Fanuc TP program (LS listing): FM142654.ls

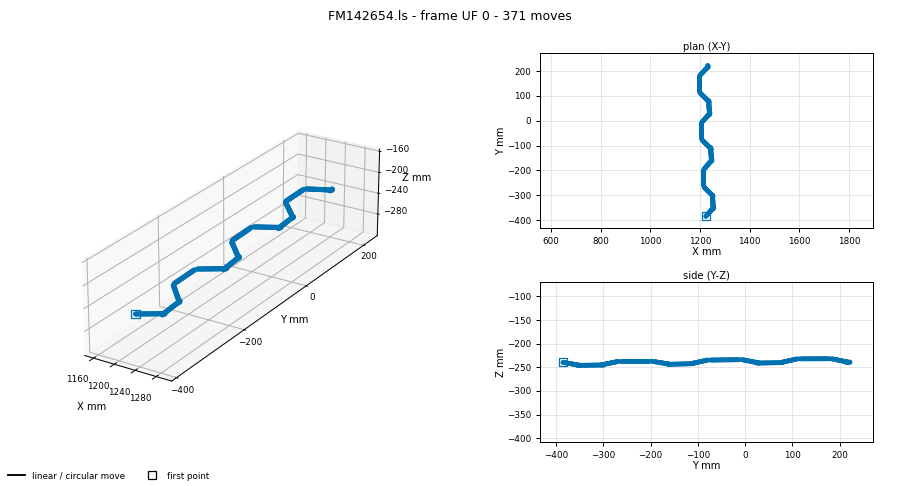
[picture p0: tool path of FM142654.ls in frame UF 0, 371 of 371 moves have a stored position in this frame; points joined in program order, loops and branches not executed]
/PROG  FM142654
/ATTR
OWNER		= MNEDITOR;
COMMENT		= "Auto FANUC move";
PROG_SIZE	= 0;
CREATE		= DATE 26-05-06  TIME 14:26:54;
MODIFIED	= DATE 26-05-06  TIME 14:26:54;
FILE_NAME	= ;
VERSION		= 0;
LINE_COUNT	= 376;
MEMORY_SIZE	= 0;
PROTECT		= READ_WRITE;
TCD:  STACK_SIZE	= 0,
      TASK_PRIORITY	= 50,
      TIME_SLICE	= 0,
      BUSY_LAMP_OFF	= 0,
      ABORT_REQUEST	= 0,
      PAUSE_REQUEST	= 0;
DEFAULT_GROUP	= 1,*,*,*,*;
CONTROL_CODE	= 00000000 00000000;
/MN
   1:  UFRAME_NUM=0 ;
   2:  UTOOL_NUM=1 ;
   3:  R[93]=10 ;
   4:  L P[1] 7mm/sec FINE ;
   5:  L P[2] 7mm/sec CNT50 ;
   6:  L P[3] 7mm/sec CNT50 ;
   7:  L P[4] 7mm/sec CNT50 ;
   8:  L P[5] 7mm/sec CNT50 ;
   9:  L P[6] 7mm/sec CNT50 ;
  10:  L P[7] 7mm/sec CNT50 ;
  11:  L P[8] 7mm/sec CNT50 ;
  12:  L P[9] 7mm/sec CNT50 ;
  13:  L P[10] 7mm/sec CNT50 ;
  14:  L P[11] 7mm/sec CNT50 ;
  15:  L P[12] 7mm/sec CNT50 ;
  16:  L P[13] 7mm/sec CNT50 ;
  17:  L P[14] 7mm/sec CNT50 ;
  18:  L P[15] 7mm/sec CNT50 ;
  19:  L P[16] 7mm/sec CNT50 ;
  20:  L P[17] 7mm/sec CNT50 ;
  21:  L P[18] 7mm/sec CNT50 ;
  22:  L P[19] 7mm/sec CNT50 ;
  23:  L P[20] 7mm/sec CNT50 ;
  24:  L P[21] 7mm/sec CNT50 ;
  25:  L P[22] 7mm/sec CNT50 ;
  26:  L P[23] 7mm/sec CNT50 ;
  27:  L P[24] 7mm/sec CNT50 ;
  28:  L P[25] 7mm/sec CNT50 ;
  29:  L P[26] 7mm/sec CNT50 ;
  30:  L P[27] 7mm/sec CNT50 ;
  31:  L P[28] 7mm/sec CNT50 ;
  32:  L P[29] 7mm/sec CNT50 ;
  33:  L P[30] 7mm/sec CNT50 ;
  34:  L P[31] 7mm/sec CNT50 ;
  35:  L P[32] 7mm/sec CNT50 ;
  36:  L P[33] 7mm/sec CNT50 ;
  37:  L P[34] 7mm/sec CNT50 ;
  38:  L P[35] 7mm/sec CNT50 ;
  39:  L P[36] 7mm/sec CNT50 ;
  40:  L P[37] 7mm/sec CNT50 ;
  41:  L P[38] 7mm/sec CNT50 ;
  42:  L P[39] 7mm/sec CNT50 ;
  43:  L P[40] 7mm/sec CNT50 ;
  44:  L P[41] 7mm/sec CNT50 ;
  45:  L P[42] 7mm/sec CNT50 ;
  46:  L P[43] 7mm/sec CNT50 ;
  47:  L P[44] 7mm/sec CNT50 ;
  48:  L P[45] 7mm/sec CNT50 ;
  49:  L P[46] 7mm/sec CNT50 ;
  50:  L P[47] 7mm/sec CNT50 ;
  51:  L P[48] 7mm/sec CNT50 ;
  52:  L P[49] 7mm/sec CNT50 ;
  53:  L P[50] 7mm/sec CNT50 ;
  54:  L P[51] 7mm/sec CNT50 ;
  55:  L P[52] 7mm/sec CNT50 ;
  56:  L P[53] 7mm/sec CNT50 ;
  57:  L P[54] 7mm/sec CNT50 ;
  58:  L P[55] 7mm/sec CNT50 ;
  59:  L P[56] 7mm/sec CNT50 ;
  60:  L P[57] 7mm/sec CNT50 ;
  61:  L P[58] 7mm/sec CNT50 ;
  62:  L P[59] 7mm/sec CNT50 ;
  63:  L P[60] 7mm/sec CNT50 ;
  64:  L P[61] 7mm/sec CNT50 ;
  65:  L P[62] 7mm/sec CNT50 ;
  66:  L P[63] 7mm/sec CNT50 ;
  67:  L P[64] 7mm/sec CNT50 ;
  68:  L P[65] 7mm/sec CNT50 ;
  69:  L P[66] 7mm/sec CNT50 ;
  70:  L P[67] 7mm/sec CNT50 ;
  71:  L P[68] 7mm/sec CNT50 ;
  72:  L P[69] 7mm/sec CNT50 ;
  73:  L P[70] 7mm/sec CNT50 ;
  74:  L P[71] 7mm/sec CNT50 ;
  75:  L P[72] 7mm/sec CNT50 ;
  76:  L P[73] 7mm/sec CNT50 ;
  77:  L P[74] 7mm/sec CNT50 ;
  78:  L P[75] 7mm/sec CNT50 ;
  79:  L P[76] 7mm/sec CNT50 ;
  80:  L P[77] 7mm/sec CNT50 ;
  81:  L P[78] 7mm/sec CNT50 ;
  82:  L P[79] 7mm/sec CNT50 ;
  83:  L P[80] 7mm/sec CNT50 ;
  84:  L P[81] 7mm/sec CNT50 ;
  85:  L P[82] 7mm/sec CNT50 ;
  86:  L P[83] 7mm/sec CNT50 ;
  87:  L P[84] 7mm/sec CNT50 ;
  88:  L P[85] 7mm/sec CNT50 ;
  89:  L P[86] 7mm/sec CNT50 ;
  90:  L P[87] 7mm/sec CNT50 ;
  91:  L P[88] 7mm/sec CNT50 ;
  92:  L P[89] 7mm/sec CNT50 ;
  93:  L P[90] 7mm/sec CNT50 ;
  94:  L P[91] 7mm/sec CNT50 ;
  95:  L P[92] 7mm/sec CNT50 ;
  96:  L P[93] 7mm/sec CNT50 ;
  97:  L P[94] 7mm/sec CNT50 ;
  98:  L P[95] 7mm/sec CNT50 ;
  99:  L P[96] 7mm/sec CNT50 ;
 100:  L P[97] 7mm/sec CNT50 ;
 101:  L P[98] 7mm/sec CNT50 ;
 102:  L P[99] 7mm/sec CNT50 ;
 103:  L P[100] 7mm/sec CNT50 ;
 104:  L P[101] 7mm/sec CNT50 ;
 105:  L P[102] 7mm/sec CNT50 ;
 106:  L P[103] 7mm/sec CNT50 ;
 107:  L P[104] 7mm/sec CNT50 ;
 108:  L P[105] 7mm/sec CNT50 ;
 109:  L P[106] 7mm/sec CNT50 ;
 110:  L P[107] 7mm/sec CNT50 ;
 111:  L P[108] 7mm/sec CNT50 ;
 112:  L P[109] 7mm/sec CNT50 ;
 113:  L P[110] 7mm/sec CNT50 ;
 114:  L P[111] 7mm/sec CNT50 ;
 115:  L P[112] 7mm/sec CNT50 ;
 116:  L P[113] 7mm/sec CNT50 ;
 117:  L P[114] 7mm/sec CNT50 ;
 118:  L P[115] 7mm/sec CNT50 ;
 119:  L P[116] 7mm/sec CNT50 ;
 120:  L P[117] 7mm/sec CNT50 ;
 121:  L P[118] 7mm/sec CNT50 ;
 122:  L P[119] 7mm/sec CNT50 ;
 123:  L P[120] 7mm/sec CNT50 ;
 124:  L P[121] 7mm/sec CNT50 ;
 125:  L P[122] 7mm/sec CNT50 ;
 126:  L P[123] 7mm/sec CNT50 ;
 127:  L P[124] 7mm/sec CNT50 ;
 128:  L P[125] 7mm/sec CNT50 ;
 129:  L P[126] 7mm/sec CNT50 ;
 130:  L P[127] 7mm/sec CNT50 ;
 131:  L P[128] 7mm/sec CNT50 ;
 132:  L P[129] 7mm/sec CNT50 ;
 133:  L P[130] 7mm/sec CNT50 ;
 134:  L P[131] 7mm/sec CNT50 ;
 135:  L P[132] 7mm/sec CNT50 ;
 136:  L P[133] 7mm/sec CNT50 ;
 137:  L P[134] 7mm/sec CNT50 ;
 138:  L P[135] 7mm/sec CNT50 ;
 139:  L P[136] 7mm/sec CNT50 ;
 140:  L P[137] 7mm/sec CNT50 ;
 141:  L P[138] 7mm/sec CNT50 ;
 142:  L P[139] 7mm/sec CNT50 ;
 143:  L P[140] 7mm/sec CNT50 ;
 144:  L P[141] 7mm/sec CNT50 ;
 145:  L P[142] 7mm/sec CNT50 ;
 146:  L P[143] 7mm/sec CNT50 ;
 147:  L P[144] 7mm/sec CNT50 ;
 148:  L P[145] 7mm/sec CNT50 ;
 149:  L P[146] 7mm/sec CNT50 ;
 150:  L P[147] 7mm/sec CNT50 ;
 151:  L P[148] 7mm/sec CNT50 ;
 152:  L P[149] 7mm/sec CNT50 ;
 153:  L P[150] 7mm/sec CNT50 ;
 154:  L P[151] 7mm/sec CNT50 ;
 155:  L P[152] 7mm/sec CNT50 ;
 156:  L P[153] 7mm/sec CNT50 ;
 157:  L P[154] 7mm/sec CNT50 ;
 158:  L P[155] 7mm/sec CNT50 ;
 159:  L P[156] 7mm/sec CNT50 ;
 160:  L P[157] 7mm/sec CNT50 ;
 161:  L P[158] 7mm/sec CNT50 ;
 162:  L P[159] 7mm/sec CNT50 ;
 163:  L P[160] 7mm/sec CNT50 ;
 164:  L P[161] 7mm/sec CNT50 ;
 165:  L P[162] 7mm/sec CNT50 ;
 166:  L P[163] 7mm/sec CNT50 ;
 167:  L P[164] 7mm/sec CNT50 ;
 168:  L P[165] 7mm/sec CNT50 ;
 169:  L P[166] 7mm/sec CNT50 ;
 170:  L P[167] 7mm/sec CNT50 ;
 171:  L P[168] 7mm/sec CNT50 ;
 172:  L P[169] 7mm/sec CNT50 ;
 173:  L P[170] 7mm/sec CNT50 ;
 174:  L P[171] 7mm/sec CNT50 ;
 175:  L P[172] 7mm/sec CNT50 ;
 176:  L P[173] 7mm/sec CNT50 ;
 177:  L P[174] 7mm/sec CNT50 ;
 178:  L P[175] 7mm/sec CNT50 ;
 179:  L P[176] 7mm/sec CNT50 ;
 180:  L P[177] 7mm/sec CNT50 ;
 181:  L P[178] 7mm/sec CNT50 ;
 182:  L P[179] 7mm/sec CNT50 ;
 183:  L P[180] 7mm/sec CNT50 ;
 184:  L P[181] 7mm/sec CNT50 ;
 185:  L P[182] 7mm/sec CNT50 ;
 186:  L P[183] 7mm/sec CNT50 ;
 187:  L P[184] 7mm/sec CNT50 ;
 188:  L P[185] 7mm/sec CNT50 ;
 189:  L P[186] 7mm/sec CNT50 ;
 190:  L P[187] 7mm/sec CNT50 ;
 191:  L P[188] 7mm/sec CNT50 ;
 192:  L P[189] 7mm/sec CNT50 ;
 193:  L P[190] 7mm/sec CNT50 ;
 194:  L P[191] 7mm/sec CNT50 ;
 195:  L P[192] 7mm/sec CNT50 ;
 196:  L P[193] 7mm/sec CNT50 ;
 197:  L P[194] 7mm/sec CNT50 ;
 198:  L P[195] 7mm/sec CNT50 ;
 199:  L P[196] 7mm/sec CNT50 ;
 200:  L P[197] 7mm/sec CNT50 ;
 201:  L P[198] 7mm/sec CNT50 ;
 202:  L P[199] 7mm/sec CNT50 ;
 203:  L P[200] 7mm/sec CNT50 ;
 204:  L P[201] 7mm/sec CNT50 ;
 205:  L P[202] 7mm/sec CNT50 ;
 206:  L P[203] 7mm/sec CNT50 ;
 207:  L P[204] 7mm/sec CNT50 ;
 208:  L P[205] 7mm/sec CNT50 ;
 209:  L P[206] 7mm/sec CNT50 ;
 210:  L P[207] 7mm/sec CNT50 ;
 211:  L P[208] 7mm/sec CNT50 ;
 212:  L P[209] 7mm/sec CNT50 ;
 213:  L P[210] 7mm/sec CNT50 ;
 214:  L P[211] 7mm/sec CNT50 ;
 215:  L P[212] 7mm/sec CNT50 ;
 216:  L P[213] 7mm/sec CNT50 ;
 217:  L P[214] 7mm/sec CNT50 ;
 218:  L P[215] 7mm/sec CNT50 ;
 219:  L P[216] 7mm/sec CNT50 ;
 220:  L P[217] 7mm/sec CNT50 ;
 221:  L P[218] 7mm/sec CNT50 ;
 222:  L P[219] 7mm/sec CNT50 ;
 223:  L P[220] 7mm/sec CNT50 ;
 224:  L P[221] 7mm/sec CNT50 ;
 225:  L P[222] 7mm/sec CNT50 ;
 226:  L P[223] 7mm/sec CNT50 ;
 227:  L P[224] 7mm/sec CNT50 ;
 228:  L P[225] 7mm/sec CNT50 ;
 229:  L P[226] 7mm/sec CNT50 ;
 230:  L P[227] 7mm/sec CNT50 ;
 231:  L P[228] 7mm/sec CNT50 ;
 232:  L P[229] 7mm/sec CNT50 ;
 233:  L P[230] 7mm/sec CNT50 ;
 234:  L P[231] 7mm/sec CNT50 ;
 235:  L P[232] 7mm/sec CNT50 ;
 236:  L P[233] 7mm/sec CNT50 ;
 237:  L P[234] 7mm/sec CNT50 ;
 238:  L P[235] 7mm/sec CNT50 ;
 239:  L P[236] 7mm/sec CNT50 ;
 240:  L P[237] 7mm/sec CNT50 ;
 241:  L P[238] 7mm/sec CNT50 ;
 242:  L P[239] 7mm/sec CNT50 ;
 243:  L P[240] 7mm/sec CNT50 ;
 244:  L P[241] 7mm/sec CNT50 ;
 245:  L P[242] 7mm/sec CNT50 ;
 246:  L P[243] 7mm/sec CNT50 ;
 247:  L P[244] 7mm/sec CNT50 ;
 248:  L P[245] 7mm/sec CNT50 ;
 249:  L P[246] 7mm/sec CNT50 ;
 250:  L P[247] 7mm/sec CNT50 ;
 251:  L P[248] 7mm/sec CNT50 ;
 252:  L P[249] 7mm/sec CNT50 ;
 253:  L P[250] 7mm/sec CNT50 ;
 254:  L P[251] 7mm/sec CNT50 ;
 255:  L P[252] 7mm/sec CNT50 ;
 256:  L P[253] 7mm/sec CNT50 ;
 257:  L P[254] 7mm/sec CNT50 ;
 258:  L P[255] 7mm/sec CNT50 ;
 259:  L P[256] 7mm/sec CNT50 ;
 260:  L P[257] 7mm/sec CNT50 ;
 261:  L P[258] 7mm/sec CNT50 ;
 262:  L P[259] 7mm/sec CNT50 ;
 263:  L P[260] 7mm/sec CNT50 ;
 264:  L P[261] 7mm/sec CNT50 ;
 265:  L P[262] 7mm/sec CNT50 ;
 266:  L P[263] 7mm/sec CNT50 ;
 267:  L P[264] 7mm/sec CNT50 ;
 268:  L P[265] 7mm/sec CNT50 ;
 269:  L P[266] 7mm/sec CNT50 ;
 270:  L P[267] 7mm/sec CNT50 ;
 271:  L P[268] 7mm/sec CNT50 ;
 272:  L P[269] 7mm/sec CNT50 ;
 273:  L P[270] 7mm/sec CNT50 ;
 274:  L P[271] 7mm/sec CNT50 ;
 275:  L P[272] 7mm/sec CNT50 ;
 276:  L P[273] 7mm/sec CNT50 ;
 277:  L P[274] 7mm/sec CNT50 ;
 278:  L P[275] 7mm/sec CNT50 ;
 279:  L P[276] 7mm/sec CNT50 ;
 280:  L P[277] 7mm/sec CNT50 ;
 281:  L P[278] 7mm/sec CNT50 ;
 282:  L P[279] 7mm/sec CNT50 ;
 283:  L P[280] 7mm/sec CNT50 ;
 284:  L P[281] 7mm/sec CNT50 ;
 285:  L P[282] 7mm/sec CNT50 ;
 286:  L P[283] 7mm/sec CNT50 ;
 287:  L P[284] 7mm/sec CNT50 ;
 288:  L P[285] 7mm/sec CNT50 ;
 289:  L P[286] 7mm/sec CNT50 ;
 290:  L P[287] 7mm/sec CNT50 ;
 291:  L P[288] 7mm/sec CNT50 ;
 292:  L P[289] 7mm/sec CNT50 ;
 293:  L P[290] 7mm/sec CNT50 ;
 294:  L P[291] 7mm/sec CNT50 ;
 295:  L P[292] 7mm/sec CNT50 ;
 296:  L P[293] 7mm/sec CNT50 ;
 297:  L P[294] 7mm/sec CNT50 ;
 298:  L P[295] 7mm/sec CNT50 ;
 299:  L P[296] 7mm/sec CNT50 ;
 300:  L P[297] 7mm/sec CNT50 ;
 301:  L P[298] 7mm/sec CNT50 ;
 302:  L P[299] 7mm/sec CNT50 ;
 303:  L P[300] 7mm/sec CNT50 ;
 304:  L P[301] 7mm/sec CNT50 ;
 305:  L P[302] 7mm/sec CNT50 ;
 306:  L P[303] 7mm/sec CNT50 ;
 307:  L P[304] 7mm/sec CNT50 ;
 308:  L P[305] 7mm/sec CNT50 ;
 309:  L P[306] 7mm/sec CNT50 ;
 310:  L P[307] 7mm/sec CNT50 ;
 311:  L P[308] 7mm/sec CNT50 ;
 312:  L P[309] 7mm/sec CNT50 ;
 313:  L P[310] 7mm/sec CNT50 ;
 314:  L P[311] 7mm/sec CNT50 ;
 315:  L P[312] 7mm/sec CNT50 ;
 316:  L P[313] 7mm/sec CNT50 ;
 317:  L P[314] 7mm/sec CNT50 ;
 318:  L P[315] 7mm/sec CNT50 ;
 319:  L P[316] 7mm/sec CNT50 ;
 320:  L P[317] 7mm/sec CNT50 ;
 321:  L P[318] 7mm/sec CNT50 ;
 322:  L P[319] 7mm/sec CNT50 ;
 323:  L P[320] 7mm/sec CNT50 ;
 324:  L P[321] 7mm/sec CNT50 ;
 325:  L P[322] 7mm/sec CNT50 ;
 326:  L P[323] 7mm/sec CNT50 ;
 327:  L P[324] 7mm/sec CNT50 ;
 328:  L P[325] 7mm/sec CNT50 ;
 329:  L P[326] 7mm/sec CNT50 ;
 330:  L P[327] 7mm/sec CNT50 ;
 331:  L P[328] 7mm/sec CNT50 ;
 332:  L P[329] 7mm/sec CNT50 ;
 333:  L P[330] 7mm/sec CNT50 ;
 334:  L P[331] 7mm/sec CNT50 ;
 335:  L P[332] 7mm/sec CNT50 ;
 336:  L P[333] 7mm/sec CNT50 ;
 337:  L P[334] 7mm/sec CNT50 ;
 338:  L P[335] 7mm/sec CNT50 ;
 339:  L P[336] 7mm/sec CNT50 ;
 340:  L P[337] 7mm/sec CNT50 ;
 341:  L P[338] 7mm/sec CNT50 ;
 342:  L P[339] 7mm/sec CNT50 ;
 343:  L P[340] 7mm/sec CNT50 ;
 344:  L P[341] 7mm/sec CNT50 ;
 345:  L P[342] 7mm/sec CNT50 ;
 346:  L P[343] 7mm/sec CNT50 ;
 347:  L P[344] 7mm/sec CNT50 ;
 348:  L P[345] 7mm/sec CNT50 ;
 349:  L P[346] 7mm/sec CNT50 ;
 350:  L P[347] 7mm/sec CNT50 ;
 351:  L P[348] 7mm/sec CNT50 ;
 352:  L P[349] 7mm/sec CNT50 ;
 353:  L P[350] 7mm/sec CNT50 ;
 354:  L P[351] 7mm/sec CNT50 ;
 355:  L P[352] 7mm/sec CNT50 ;
 356:  L P[353] 7mm/sec CNT50 ;
 357:  L P[354] 7mm/sec CNT50 ;
 358:  L P[355] 7mm/sec CNT50 ;
 359:  L P[356] 7mm/sec CNT50 ;
 360:  L P[357] 7mm/sec CNT50 ;
 361:  L P[358] 7mm/sec CNT50 ;
 362:  L P[359] 7mm/sec CNT50 ;
 363:  L P[360] 7mm/sec CNT50 ;
 364:  L P[361] 7mm/sec CNT50 ;
 365:  L P[362] 7mm/sec CNT50 ;
 366:  L P[363] 7mm/sec CNT50 ;
 367:  L P[364] 7mm/sec CNT50 ;
 368:  L P[365] 7mm/sec CNT50 ;
 369:  L P[366] 7mm/sec CNT50 ;
 370:  L P[367] 7mm/sec CNT50 ;
 371:  L P[368] 7mm/sec CNT50 ;
 372:  L P[369] 7mm/sec CNT50 ;
 373:  L P[370] 7mm/sec CNT50 ;
 374:  L P[371] 7mm/sec FINE ;
 375:  R[93]=1 ;
 376:  END ;
/POS
P[1]{
   GP1:
	UF : 0, UT : 1,		CONFIG : 'N U T, 0, 0, 0',
	X = 1223.194  mm,	Y = -385.306  mm,	Z = -239.653  mm,
	W = 0.000 deg,	P = 30.000 deg,	R = 138.708 deg
};
P[2]{
   GP1:
	UF : 0, UT : 1,		CONFIG : 'N U T, 0, 0, 0',
	X = 1224.503  mm,	Y = -383.816  mm,	Z = -239.910  mm,
	W = 0.000 deg,	P = 30.000 deg,	R = 138.708 deg
};
P[3]{
   GP1:
	UF : 0, UT : 1,		CONFIG : 'N U T, 0, 0, 0',
	X = 1225.812  mm,	Y = -382.326  mm,	Z = -240.167  mm,
	W = 0.000 deg,	P = 30.000 deg,	R = 138.708 deg
};
P[4]{
   GP1:
	UF : 0, UT : 1,		CONFIG : 'N U T, 0, 0, 0',
	X = 1227.120  mm,	Y = -380.835  mm,	Z = -240.424  mm,
	W = 0.000 deg,	P = 30.000 deg,	R = 138.708 deg
};
P[5]{
   GP1:
	UF : 0, UT : 1,		CONFIG : 'N U T, 0, 0, 0',
	X = 1228.429  mm,	Y = -379.345  mm,	Z = -240.682  mm,
	W = 0.000 deg,	P = 30.000 deg,	R = 138.708 deg
};
P[6]{
   GP1:
	UF : 0, UT : 1,		CONFIG : 'N U T, 0, 0, 0',
	X = 1229.738  mm,	Y = -377.855  mm,	Z = -240.939  mm,
	W = 0.000 deg,	P = 30.000 deg,	R = 138.708 deg
};
P[7]{
   GP1:
	UF : 0, UT : 1,		CONFIG : 'N U T, 0, 0, 0',
	X = 1231.047  mm,	Y = -376.365  mm,	Z = -241.196  mm,
	W = 0.000 deg,	P = 30.000 deg,	R = 138.708 deg
};
P[8]{
   GP1:
	UF : 0, UT : 1,		CONFIG : 'N U T, 0, 0, 0',
	X = 1232.356  mm,	Y = -374.874  mm,	Z = -241.453  mm,
	W = 0.000 deg,	P = 30.000 deg,	R = 138.708 deg
};
P[9]{
   GP1:
	UF : 0, UT : 1,		CONFIG : 'N U T, 0, 0, 0',
	X = 1233.665  mm,	Y = -373.384  mm,	Z = -241.710  mm,
	W = 0.000 deg,	P = 30.000 deg,	R = 138.708 deg
};
P[10]{
   GP1:
	UF : 0, UT : 1,		CONFIG : 'N U T, 0, 0, 0',
	X = 1234.973  mm,	Y = -371.894  mm,	Z = -241.967  mm,
	W = 0.000 deg,	P = 30.000 deg,	R = 138.708 deg
};
P[11]{
   GP1:
	UF : 0, UT : 1,		CONFIG : 'N U T, 0, 0, 0',
	X = 1236.282  mm,	Y = -370.404  mm,	Z = -242.225  mm,
	W = 0.000 deg,	P = 30.000 deg,	R = 138.708 deg
};
P[12]{
   GP1:
	UF : 0, UT : 1,		CONFIG : 'N U T, 0, 0, 0',
	X = 1237.591  mm,	Y = -368.913  mm,	Z = -242.482  mm,
	W = 0.000 deg,	P = 30.000 deg,	R = 138.708 deg
};
P[13]{
   GP1:
	UF : 0, UT : 1,		CONFIG : 'N U T, 0, 0, 0',
	X = 1238.900  mm,	Y = -367.423  mm,	Z = -242.739  mm,
	W = 0.000 deg,	P = 30.000 deg,	R = 138.708 deg
};
P[14]{
   GP1:
	UF : 0, UT : 1,		CONFIG : 'N U T, 0, 0, 0',
	X = 1240.209  mm,	Y = -365.933  mm,	Z = -242.996  mm,
	W = 0.000 deg,	P = 30.000 deg,	R = 138.708 deg
};
P[15]{
   GP1:
	UF : 0, UT : 1,		CONFIG : 'N U T, 0, 0, 0',
	X = 1241.518  mm,	Y = -364.443  mm,	Z = -243.253  mm,
	W = 0.000 deg,	P = 30.000 deg,	R = 138.708 deg
};
P[16]{
   GP1:
	UF : 0, UT : 1,		CONFIG : 'N U T, 0, 0, 0',
	X = 1242.826  mm,	Y = -362.952  mm,	Z = -243.510  mm,
	W = 0.000 deg,	P = 30.000 deg,	R = 138.708 deg
};
P[17]{
   GP1:
	UF : 0, UT : 1,		CONFIG : 'N U T, 0, 0, 0',
	X = 1244.135  mm,	Y = -361.462  mm,	Z = -243.767  mm,
	W = 0.000 deg,	P = 30.000 deg,	R = 138.708 deg
};
P[18]{
   GP1:
	UF : 0, UT : 1,		CONFIG : 'N U T, 0, 0, 0',
	X = 1245.444  mm,	Y = -359.972  mm,	Z = -244.025  mm,
	W = 0.000 deg,	P = 30.000 deg,	R = 138.708 deg
};
P[19]{
   GP1:
	UF : 0, UT : 1,		CONFIG : 'N U T, 0, 0, 0',
	X = 1246.753  mm,	Y = -358.482  mm,	Z = -244.282  mm,
	W = 0.000 deg,	P = 30.000 deg,	R = 138.708 deg
};
P[20]{
   GP1:
	UF : 0, UT : 1,		CONFIG : 'N U T, 0, 0, 0',
	X = 1248.062  mm,	Y = -356.991  mm,	Z = -244.539  mm,
	W = 0.000 deg,	P = 30.000 deg,	R = 138.708 deg
};
P[21]{
   GP1:
	UF : 0, UT : 1,		CONFIG : 'N U T, 0, 0, 0',
	X = 1249.371  mm,	Y = -355.501  mm,	Z = -244.796  mm,
	W = 0.000 deg,	P = 30.000 deg,	R = 147.583 deg
};
P[22]{
   GP1:
	UF : 0, UT : 1,		CONFIG : 'N U T, 0, 0, 0',
	X = 1250.679  mm,	Y = -354.011  mm,	Z = -245.053  mm,
	W = 0.000 deg,	P = 30.000 deg,	R = 156.458 deg
};
P[23]{
   GP1:
	UF : 0, UT : 1,		CONFIG : 'N U T, 0, 0, 0',
	X = 1251.988  mm,	Y = -352.521  mm,	Z = -245.310  mm,
	W = 0.000 deg,	P = 30.000 deg,	R = 165.333 deg
};
P[24]{
   GP1:
	UF : 0, UT : 1,		CONFIG : 'N U T, 0, 0, 0',
	X = 1253.297  mm,	Y = -351.030  mm,	Z = -245.568  mm,
	W = 0.000 deg,	P = 30.000 deg,	R = 174.208 deg
};
P[25]{
   GP1:
	UF : 0, UT : 1,		CONFIG : 'N U T, 0, 0, 0',
	X = 1254.606  mm,	Y = -349.540  mm,	Z = -245.825  mm,
	W = 0.000 deg,	P = 30.000 deg,	R = -176.917 deg
};
P[26]{
   GP1:
	UF : 0, UT : 1,		CONFIG : 'N U T, 0, 0, 0',
	X = 1254.120  mm,	Y = -350.543  mm,	Z = -245.999  mm,
	W = 0.000 deg,	P = 30.000 deg,	R = -176.917 deg
};
P[27]{
   GP1:
	UF : 0, UT : 1,		CONFIG : 'N U T, 0, 0, 0',
	X = 1252.987  mm,	Y = -355.024  mm,	Z = -245.989  mm,
	W = 0.000 deg,	P = 30.000 deg,	R = -176.917 deg
};
P[28]{
   GP1:
	UF : 0, UT : 1,		CONFIG : 'N U T, 0, 0, 0',
	X = 1252.879  mm,	Y = -353.027  mm,	Z = -245.958  mm,
	W = 0.000 deg,	P = 30.000 deg,	R = -176.917 deg
};
P[29]{
   GP1:
	UF : 0, UT : 1,		CONFIG : 'N U T, 0, 0, 0',
	X = 1252.772  mm,	Y = -351.030  mm,	Z = -245.926  mm,
	W = 0.000 deg,	P = 30.000 deg,	R = -176.917 deg
};
P[30]{
   GP1:
	UF : 0, UT : 1,		CONFIG : 'N U T, 0, 0, 0',
	X = 1252.664  mm,	Y = -349.033  mm,	Z = -245.895  mm,
	W = 0.000 deg,	P = 30.000 deg,	R = -176.917 deg
};
P[31]{
   GP1:
	UF : 0, UT : 1,		CONFIG : 'N U T, 0, 0, 0',
	X = 1252.557  mm,	Y = -347.036  mm,	Z = -245.863  mm,
	W = 0.000 deg,	P = 30.000 deg,	R = -176.917 deg
};
P[32]{
   GP1:
	UF : 0, UT : 1,		CONFIG : 'N U T, 0, 0, 0',
	X = 1252.449  mm,	Y = -345.039  mm,	Z = -245.832  mm,
	W = 0.000 deg,	P = 30.000 deg,	R = -176.917 deg
};
P[33]{
   GP1:
	UF : 0, UT : 1,		CONFIG : 'N U T, 0, 0, 0',
	X = 1252.342  mm,	Y = -343.042  mm,	Z = -245.801  mm,
	W = 0.000 deg,	P = 30.000 deg,	R = -176.917 deg
};
P[34]{
   GP1:
	UF : 0, UT : 1,		CONFIG : 'N U T, 0, 0, 0',
	X = 1252.234  mm,	Y = -341.046  mm,	Z = -245.769  mm,
	W = 0.000 deg,	P = 30.000 deg,	R = -176.917 deg
};
P[35]{
   GP1:
	UF : 0, UT : 1,		CONFIG : 'N U T, 0, 0, 0',
	X = 1252.126  mm,	Y = -339.049  mm,	Z = -245.738  mm,
	W = 0.000 deg,	P = 30.000 deg,	R = -176.917 deg
};
P[36]{
   GP1:
	UF : 0, UT : 1,		CONFIG : 'N U T, 0, 0, 0',
	X = 1252.019  mm,	Y = -337.052  mm,	Z = -245.706  mm,
	W = 0.000 deg,	P = 30.000 deg,	R = -176.917 deg
};
P[37]{
   GP1:
	UF : 0, UT : 1,		CONFIG : 'N U T, 0, 0, 0',
	X = 1251.911  mm,	Y = -335.055  mm,	Z = -245.675  mm,
	W = 0.000 deg,	P = 30.000 deg,	R = -176.917 deg
};
P[38]{
   GP1:
	UF : 0, UT : 1,		CONFIG : 'N U T, 0, 0, 0',
	X = 1251.804  mm,	Y = -333.058  mm,	Z = -245.644  mm,
	W = 0.000 deg,	P = 30.000 deg,	R = -176.917 deg
};
P[39]{
   GP1:
	UF : 0, UT : 1,		CONFIG : 'N U T, 0, 0, 0',
	X = 1251.696  mm,	Y = -331.061  mm,	Z = -245.612  mm,
	W = 0.000 deg,	P = 30.000 deg,	R = -176.917 deg
};
P[40]{
   GP1:
	UF : 0, UT : 1,		CONFIG : 'N U T, 0, 0, 0',
	X = 1251.589  mm,	Y = -329.064  mm,	Z = -245.581  mm,
	W = 0.000 deg,	P = 30.000 deg,	R = -176.917 deg
};
P[41]{
   GP1:
	UF : 0, UT : 1,		CONFIG : 'N U T, 0, 0, 0',
	X = 1251.481  mm,	Y = -327.068  mm,	Z = -245.549  mm,
	W = 0.000 deg,	P = 30.000 deg,	R = -176.917 deg
};
P[42]{
   GP1:
	UF : 0, UT : 1,		CONFIG : 'N U T, 0, 0, 0',
	X = 1251.374  mm,	Y = -325.071  mm,	Z = -245.518  mm,
	W = 0.000 deg,	P = 30.000 deg,	R = -176.917 deg
};
P[43]{
   GP1:
	UF : 0, UT : 1,		CONFIG : 'N U T, 0, 0, 0',
	X = 1251.266  mm,	Y = -323.074  mm,	Z = -245.487  mm,
	W = 0.000 deg,	P = 30.000 deg,	R = -176.917 deg
};
P[44]{
   GP1:
	UF : 0, UT : 1,		CONFIG : 'N U T, 0, 0, 0',
	X = 1251.158  mm,	Y = -321.077  mm,	Z = -245.455  mm,
	W = 0.000 deg,	P = 30.000 deg,	R = -176.917 deg
};
P[45]{
   GP1:
	UF : 0, UT : 1,		CONFIG : 'N U T, 0, 0, 0',
	X = 1251.051  mm,	Y = -319.080  mm,	Z = -245.424  mm,
	W = 0.000 deg,	P = 30.000 deg,	R = -176.917 deg
};
P[46]{
   GP1:
	UF : 0, UT : 1,		CONFIG : 'N U T, 0, 0, 0',
	X = 1250.943  mm,	Y = -317.083  mm,	Z = -245.392  mm,
	W = 0.000 deg,	P = 30.000 deg,	R = -176.917 deg
};
P[47]{
   GP1:
	UF : 0, UT : 1,		CONFIG : 'N U T, 0, 0, 0',
	X = 1250.836  mm,	Y = -315.086  mm,	Z = -245.361  mm,
	W = 0.000 deg,	P = 30.000 deg,	R = -176.917 deg
};
P[48]{
   GP1:
	UF : 0, UT : 1,		CONFIG : 'N U T, 0, 0, 0',
	X = 1250.728  mm,	Y = -313.090  mm,	Z = -245.329  mm,
	W = 0.000 deg,	P = 30.000 deg,	R = -176.917 deg
};
P[49]{
   GP1:
	UF : 0, UT : 1,		CONFIG : 'N U T, 0, 0, 0',
	X = 1250.621  mm,	Y = -311.093  mm,	Z = -245.298  mm,
	W = 0.000 deg,	P = 30.000 deg,	R = -176.917 deg
};
P[50]{
   GP1:
	UF : 0, UT : 1,		CONFIG : 'N U T, 0, 0, 0',
	X = 1250.513  mm,	Y = -309.096  mm,	Z = -245.267  mm,
	W = 0.000 deg,	P = 30.000 deg,	R = -176.917 deg
};
P[51]{
   GP1:
	UF : 0, UT : 1,		CONFIG : 'N U T, 0, 0, 0',
	X = 1250.405  mm,	Y = -307.099  mm,	Z = -245.235  mm,
	W = 0.000 deg,	P = 30.000 deg,	R = -165.910 deg
};
P[52]{
   GP1:
	UF : 0, UT : 1,		CONFIG : 'N U T, 0, 0, 0',
	X = 1250.298  mm,	Y = -305.102  mm,	Z = -245.204  mm,
	W = 0.000 deg,	P = 30.000 deg,	R = -157.583 deg
};
P[53]{
   GP1:
	UF : 0, UT : 1,		CONFIG : 'N U T, 0, 0, 0',
	X = 1250.190  mm,	Y = -303.105  mm,	Z = -245.172  mm,
	W = 0.000 deg,	P = 30.000 deg,	R = -149.255 deg
};
P[54]{
   GP1:
	UF : 0, UT : 1,		CONFIG : 'N U T, 0, 0, 0',
	X = 1250.083  mm,	Y = -301.108  mm,	Z = -245.141  mm,
	W = 0.000 deg,	P = 30.000 deg,	R = -140.928 deg
};
P[55]{
   GP1:
	UF : 0, UT : 1,		CONFIG : 'N U T, 0, 0, 0',
	X = 1249.975  mm,	Y = -299.112  mm,	Z = -245.110  mm,
	W = 0.000 deg,	P = 30.000 deg,	R = -135.281 deg
};
P[56]{
   GP1:
	UF : 0, UT : 1,		CONFIG : 'N U T, 0, 0, 0',
	X = 1250.851  mm,	Y = -301.869  mm,	Z = -245.095  mm,
	W = 0.000 deg,	P = 30.000 deg,	R = -135.281 deg
};
P[57]{
   GP1:
	UF : 0, UT : 1,		CONFIG : 'N U T, 0, 0, 0',
	X = 1252.068  mm,	Y = -303.926  mm,	Z = -244.940  mm,
	W = 0.000 deg,	P = 30.000 deg,	R = -135.281 deg
};
P[58]{
   GP1:
	UF : 0, UT : 1,		CONFIG : 'N U T, 0, 0, 0',
	X = 1250.676  mm,	Y = -302.520  mm,	Z = -244.647  mm,
	W = 0.000 deg,	P = 30.000 deg,	R = -135.281 deg
};
P[59]{
   GP1:
	UF : 0, UT : 1,		CONFIG : 'N U T, 0, 0, 0',
	X = 1249.283  mm,	Y = -301.114  mm,	Z = -244.355  mm,
	W = 0.000 deg,	P = 30.000 deg,	R = -135.281 deg
};
P[60]{
   GP1:
	UF : 0, UT : 1,		CONFIG : 'N U T, 0, 0, 0',
	X = 1247.891  mm,	Y = -299.708  mm,	Z = -244.062  mm,
	W = 0.000 deg,	P = 30.000 deg,	R = -135.281 deg
};
P[61]{
   GP1:
	UF : 0, UT : 1,		CONFIG : 'N U T, 0, 0, 0',
	X = 1246.499  mm,	Y = -298.303  mm,	Z = -243.770  mm,
	W = 0.000 deg,	P = 30.000 deg,	R = -135.281 deg
};
P[62]{
   GP1:
	UF : 0, UT : 1,		CONFIG : 'N U T, 0, 0, 0',
	X = 1245.107  mm,	Y = -296.897  mm,	Z = -243.477  mm,
	W = 0.000 deg,	P = 30.000 deg,	R = -135.281 deg
};
P[63]{
   GP1:
	UF : 0, UT : 1,		CONFIG : 'N U T, 0, 0, 0',
	X = 1243.715  mm,	Y = -295.491  mm,	Z = -243.185  mm,
	W = 0.000 deg,	P = 30.000 deg,	R = -135.281 deg
};
P[64]{
   GP1:
	UF : 0, UT : 1,		CONFIG : 'N U T, 0, 0, 0',
	X = 1242.323  mm,	Y = -294.085  mm,	Z = -242.892  mm,
	W = 0.000 deg,	P = 30.000 deg,	R = -135.281 deg
};
P[65]{
   GP1:
	UF : 0, UT : 1,		CONFIG : 'N U T, 0, 0, 0',
	X = 1240.931  mm,	Y = -292.679  mm,	Z = -242.599  mm,
	W = 0.000 deg,	P = 30.000 deg,	R = -135.281 deg
};
P[66]{
   GP1:
	UF : 0, UT : 1,		CONFIG : 'N U T, 0, 0, 0',
	X = 1239.539  mm,	Y = -291.273  mm,	Z = -242.307  mm,
	W = 0.000 deg,	P = 30.000 deg,	R = -135.281 deg
};
P[67]{
   GP1:
	UF : 0, UT : 1,		CONFIG : 'N U T, 0, 0, 0',
	X = 1238.146  mm,	Y = -289.867  mm,	Z = -242.014  mm,
	W = 0.000 deg,	P = 30.000 deg,	R = -135.281 deg
};
P[68]{
   GP1:
	UF : 0, UT : 1,		CONFIG : 'N U T, 0, 0, 0',
	X = 1236.754  mm,	Y = -288.462  mm,	Z = -241.722  mm,
	W = 0.000 deg,	P = 30.000 deg,	R = -135.281 deg
};
P[69]{
   GP1:
	UF : 0, UT : 1,		CONFIG : 'N U T, 0, 0, 0',
	X = 1235.362  mm,	Y = -287.056  mm,	Z = -241.429  mm,
	W = 0.000 deg,	P = 30.000 deg,	R = -135.281 deg
};
P[70]{
   GP1:
	UF : 0, UT : 1,		CONFIG : 'N U T, 0, 0, 0',
	X = 1233.970  mm,	Y = -285.650  mm,	Z = -241.137  mm,
	W = 0.000 deg,	P = 30.000 deg,	R = -135.281 deg
};
P[71]{
   GP1:
	UF : 0, UT : 1,		CONFIG : 'N U T, 0, 0, 0',
	X = 1232.578  mm,	Y = -284.244  mm,	Z = -240.844  mm,
	W = 0.000 deg,	P = 30.000 deg,	R = -135.281 deg
};
P[72]{
   GP1:
	UF : 0, UT : 1,		CONFIG : 'N U T, 0, 0, 0',
	X = 1231.186  mm,	Y = -282.838  mm,	Z = -240.551  mm,
	W = 0.000 deg,	P = 30.000 deg,	R = -135.281 deg
};
P[73]{
   GP1:
	UF : 0, UT : 1,		CONFIG : 'N U T, 0, 0, 0',
	X = 1229.794  mm,	Y = -281.432  mm,	Z = -240.259  mm,
	W = 0.000 deg,	P = 30.000 deg,	R = -135.281 deg
};
P[74]{
   GP1:
	UF : 0, UT : 1,		CONFIG : 'N U T, 0, 0, 0',
	X = 1228.402  mm,	Y = -280.026  mm,	Z = -239.966  mm,
	W = 0.000 deg,	P = 30.000 deg,	R = -135.281 deg
};
P[75]{
   GP1:
	UF : 0, UT : 1,		CONFIG : 'N U T, 0, 0, 0',
	X = 1227.010  mm,	Y = -278.621  mm,	Z = -239.674  mm,
	W = 0.000 deg,	P = 30.000 deg,	R = -135.281 deg
};
P[76]{
   GP1:
	UF : 0, UT : 1,		CONFIG : 'N U T, 0, 0, 0',
	X = 1225.617  mm,	Y = -277.215  mm,	Z = -239.381  mm,
	W = 0.000 deg,	P = 30.000 deg,	R = -135.281 deg
};
P[77]{
   GP1:
	UF : 0, UT : 1,		CONFIG : 'N U T, 0, 0, 0',
	X = 1224.225  mm,	Y = -275.809  mm,	Z = -239.089  mm,
	W = 0.000 deg,	P = 30.000 deg,	R = -139.912 deg
};
P[78]{
   GP1:
	UF : 0, UT : 1,		CONFIG : 'N U T, 0, 0, 0',
	X = 1222.833  mm,	Y = -274.403  mm,	Z = -238.796  mm,
	W = 0.000 deg,	P = 30.000 deg,	R = -148.662 deg
};
P[79]{
   GP1:
	UF : 0, UT : 1,		CONFIG : 'N U T, 0, 0, 0',
	X = 1221.441  mm,	Y = -272.997  mm,	Z = -238.503  mm,
	W = 0.000 deg,	P = 30.000 deg,	R = -157.411 deg
};
P[80]{
   GP1:
	UF : 0, UT : 1,		CONFIG : 'N U T, 0, 0, 0',
	X = 1220.049  mm,	Y = -271.591  mm,	Z = -238.211  mm,
	W = 0.000 deg,	P = 30.000 deg,	R = -166.161 deg
};
P[81]{
   GP1:
	UF : 0, UT : 1,		CONFIG : 'N U T, 0, 0, 0',
	X = 1218.657  mm,	Y = -270.186  mm,	Z = -237.918  mm,
	W = 0.000 deg,	P = 30.000 deg,	R = -174.911 deg
};
P[82]{
   GP1:
	UF : 0, UT : 1,		CONFIG : 'N U T, 0, 0, 0',
	X = 1216.735  mm,	Y = -268.155  mm,	Z = -237.671  mm,
	W = 0.000 deg,	P = 30.000 deg,	R = -179.030 deg
};
P[83]{
   GP1:
	UF : 0, UT : 1,		CONFIG : 'N U T, 0, 0, 0',
	X = 1214.582  mm,	Y = -261.821  mm,	Z = -237.670  mm,
	W = 0.000 deg,	P = 30.000 deg,	R = -179.030 deg
};
P[84]{
   GP1:
	UF : 0, UT : 1,		CONFIG : 'N U T, 0, 0, 0',
	X = 1214.549  mm,	Y = -259.821  mm,	Z = -237.662  mm,
	W = 0.000 deg,	P = 30.000 deg,	R = -179.030 deg
};
P[85]{
   GP1:
	UF : 0, UT : 1,		CONFIG : 'N U T, 0, 0, 0',
	X = 1214.515  mm,	Y = -257.821  mm,	Z = -237.655  mm,
	W = 0.000 deg,	P = 30.000 deg,	R = -179.030 deg
};
P[86]{
   GP1:
	UF : 0, UT : 1,		CONFIG : 'N U T, 0, 0, 0',
	X = 1214.481  mm,	Y = -255.822  mm,	Z = -237.648  mm,
	W = 0.000 deg,	P = 30.000 deg,	R = -179.030 deg
};
P[87]{
   GP1:
	UF : 0, UT : 1,		CONFIG : 'N U T, 0, 0, 0',
	X = 1214.447  mm,	Y = -253.822  mm,	Z = -237.640  mm,
	W = 0.000 deg,	P = 30.000 deg,	R = -179.030 deg
};
P[88]{
   GP1:
	UF : 0, UT : 1,		CONFIG : 'N U T, 0, 0, 0',
	X = 1214.413  mm,	Y = -251.822  mm,	Z = -237.633  mm,
	W = 0.000 deg,	P = 30.000 deg,	R = -179.030 deg
};
P[89]{
   GP1:
	UF : 0, UT : 1,		CONFIG : 'N U T, 0, 0, 0',
	X = 1214.379  mm,	Y = -249.822  mm,	Z = -237.625  mm,
	W = 0.000 deg,	P = 30.000 deg,	R = -179.030 deg
};
P[90]{
   GP1:
	UF : 0, UT : 1,		CONFIG : 'N U T, 0, 0, 0',
	X = 1214.345  mm,	Y = -247.823  mm,	Z = -237.618  mm,
	W = 0.000 deg,	P = 30.000 deg,	R = -179.030 deg
};
P[91]{
   GP1:
	UF : 0, UT : 1,		CONFIG : 'N U T, 0, 0, 0',
	X = 1214.311  mm,	Y = -245.823  mm,	Z = -237.610  mm,
	W = 0.000 deg,	P = 30.000 deg,	R = -179.030 deg
};
P[92]{
   GP1:
	UF : 0, UT : 1,		CONFIG : 'N U T, 0, 0, 0',
	X = 1214.278  mm,	Y = -243.823  mm,	Z = -237.603  mm,
	W = 0.000 deg,	P = 30.000 deg,	R = -179.030 deg
};
P[93]{
   GP1:
	UF : 0, UT : 1,		CONFIG : 'N U T, 0, 0, 0',
	X = 1214.244  mm,	Y = -241.824  mm,	Z = -237.595  mm,
	W = 0.000 deg,	P = 30.000 deg,	R = -179.030 deg
};
P[94]{
   GP1:
	UF : 0, UT : 1,		CONFIG : 'N U T, 0, 0, 0',
	X = 1214.210  mm,	Y = -239.824  mm,	Z = -237.588  mm,
	W = 0.000 deg,	P = 30.000 deg,	R = -179.030 deg
};
P[95]{
   GP1:
	UF : 0, UT : 1,		CONFIG : 'N U T, 0, 0, 0',
	X = 1214.176  mm,	Y = -237.824  mm,	Z = -237.581  mm,
	W = 0.000 deg,	P = 30.000 deg,	R = -179.030 deg
};
P[96]{
   GP1:
	UF : 0, UT : 1,		CONFIG : 'N U T, 0, 0, 0',
	X = 1214.142  mm,	Y = -235.825  mm,	Z = -237.573  mm,
	W = 0.000 deg,	P = 30.000 deg,	R = -179.030 deg
};
P[97]{
   GP1:
	UF : 0, UT : 1,		CONFIG : 'N U T, 0, 0, 0',
	X = 1214.108  mm,	Y = -233.825  mm,	Z = -237.566  mm,
	W = 0.000 deg,	P = 30.000 deg,	R = -179.030 deg
};
P[98]{
   GP1:
	UF : 0, UT : 1,		CONFIG : 'N U T, 0, 0, 0',
	X = 1214.074  mm,	Y = -231.825  mm,	Z = -237.558  mm,
	W = 0.000 deg,	P = 30.000 deg,	R = -179.030 deg
};
P[99]{
   GP1:
	UF : 0, UT : 1,		CONFIG : 'N U T, 0, 0, 0',
	X = 1214.041  mm,	Y = -229.826  mm,	Z = -237.551  mm,
	W = 0.000 deg,	P = 30.000 deg,	R = -179.030 deg
};
P[100]{
   GP1:
	UF : 0, UT : 1,		CONFIG : 'N U T, 0, 0, 0',
	X = 1214.007  mm,	Y = -227.826  mm,	Z = -237.543  mm,
	W = 0.000 deg,	P = 30.000 deg,	R = -179.030 deg
};
P[101]{
   GP1:
	UF : 0, UT : 1,		CONFIG : 'N U T, 0, 0, 0',
	X = 1213.973  mm,	Y = -225.826  mm,	Z = -237.536  mm,
	W = 0.000 deg,	P = 30.000 deg,	R = -179.030 deg
};
P[102]{
   GP1:
	UF : 0, UT : 1,		CONFIG : 'N U T, 0, 0, 0',
	X = 1213.939  mm,	Y = -223.826  mm,	Z = -237.528  mm,
	W = 0.000 deg,	P = 30.000 deg,	R = -179.030 deg
};
P[103]{
   GP1:
	UF : 0, UT : 1,		CONFIG : 'N U T, 0, 0, 0',
	X = 1213.905  mm,	Y = -221.827  mm,	Z = -237.521  mm,
	W = 0.000 deg,	P = 30.000 deg,	R = -179.030 deg
};
P[104]{
   GP1:
	UF : 0, UT : 1,		CONFIG : 'N U T, 0, 0, 0',
	X = 1213.871  mm,	Y = -219.827  mm,	Z = -237.514  mm,
	W = 0.000 deg,	P = 30.000 deg,	R = -179.030 deg
};
P[105]{
   GP1:
	UF : 0, UT : 1,		CONFIG : 'N U T, 0, 0, 0',
	X = 1213.837  mm,	Y = -217.827  mm,	Z = -237.506  mm,
	W = 0.000 deg,	P = 30.000 deg,	R = -179.030 deg
};
P[106]{
   GP1:
	UF : 0, UT : 1,		CONFIG : 'N U T, 0, 0, 0',
	X = 1213.803  mm,	Y = -215.828  mm,	Z = -237.499  mm,
	W = 0.000 deg,	P = 30.000 deg,	R = -179.030 deg
};
P[107]{
   GP1:
	UF : 0, UT : 1,		CONFIG : 'N U T, 0, 0, 0',
	X = 1213.770  mm,	Y = -213.828  mm,	Z = -237.491  mm,
	W = 0.000 deg,	P = 30.000 deg,	R = -179.030 deg
};
P[108]{
   GP1:
	UF : 0, UT : 1,		CONFIG : 'N U T, 0, 0, 0',
	X = 1213.736  mm,	Y = -211.828  mm,	Z = -237.484  mm,
	W = 0.000 deg,	P = 30.000 deg,	R = -179.030 deg
};
P[109]{
   GP1:
	UF : 0, UT : 1,		CONFIG : 'N U T, 0, 0, 0',
	X = 1213.702  mm,	Y = -209.829  mm,	Z = -237.476  mm,
	W = 0.000 deg,	P = 30.000 deg,	R = 171.466 deg
};
P[110]{
   GP1:
	UF : 0, UT : 1,		CONFIG : 'N U T, 0, 0, 0',
	X = 1213.668  mm,	Y = -207.829  mm,	Z = -237.469  mm,
	W = 0.000 deg,	P = 30.000 deg,	R = 163.237 deg
};
P[111]{
   GP1:
	UF : 0, UT : 1,		CONFIG : 'N U T, 0, 0, 0',
	X = 1213.634  mm,	Y = -205.829  mm,	Z = -237.461  mm,
	W = 0.000 deg,	P = 30.000 deg,	R = 155.008 deg
};
P[112]{
   GP1:
	UF : 0, UT : 1,		CONFIG : 'N U T, 0, 0, 0',
	X = 1213.600  mm,	Y = -203.829  mm,	Z = -237.454  mm,
	W = 0.000 deg,	P = 30.000 deg,	R = 146.778 deg
};
P[113]{
   GP1:
	UF : 0, UT : 1,		CONFIG : 'N U T, 0, 0, 0',
	X = 1213.600  mm,	Y = -201.160  mm,	Z = -237.448  mm,
	W = 0.000 deg,	P = 30.000 deg,	R = 139.825 deg
};
P[114]{
   GP1:
	UF : 0, UT : 1,		CONFIG : 'N U T, 0, 0, 0',
	X = 1216.110  mm,	Y = -195.277  mm,	Z = -237.483  mm,
	W = 0.000 deg,	P = 30.000 deg,	R = 139.825 deg
};
P[115]{
   GP1:
	UF : 0, UT : 1,		CONFIG : 'N U T, 0, 0, 0',
	X = 1217.390  mm,	Y = -193.761  mm,	Z = -237.733  mm,
	W = 0.000 deg,	P = 30.000 deg,	R = 139.825 deg
};
P[116]{
   GP1:
	UF : 0, UT : 1,		CONFIG : 'N U T, 0, 0, 0',
	X = 1218.670  mm,	Y = -192.245  mm,	Z = -237.983  mm,
	W = 0.000 deg,	P = 30.000 deg,	R = 139.825 deg
};
P[117]{
   GP1:
	UF : 0, UT : 1,		CONFIG : 'N U T, 0, 0, 0',
	X = 1219.950  mm,	Y = -190.729  mm,	Z = -238.232  mm,
	W = 0.000 deg,	P = 30.000 deg,	R = 139.825 deg
};
P[118]{
   GP1:
	UF : 0, UT : 1,		CONFIG : 'N U T, 0, 0, 0',
	X = 1221.230  mm,	Y = -189.213  mm,	Z = -238.482  mm,
	W = 0.000 deg,	P = 30.000 deg,	R = 139.825 deg
};
P[119]{
   GP1:
	UF : 0, UT : 1,		CONFIG : 'N U T, 0, 0, 0',
	X = 1222.510  mm,	Y = -187.696  mm,	Z = -238.732  mm,
	W = 0.000 deg,	P = 30.000 deg,	R = 139.825 deg
};
P[120]{
   GP1:
	UF : 0, UT : 1,		CONFIG : 'N U T, 0, 0, 0',
	X = 1223.790  mm,	Y = -186.180  mm,	Z = -238.982  mm,
	W = 0.000 deg,	P = 30.000 deg,	R = 139.825 deg
};
P[121]{
   GP1:
	UF : 0, UT : 1,		CONFIG : 'N U T, 0, 0, 0',
	X = 1225.071  mm,	Y = -184.664  mm,	Z = -239.232  mm,
	W = 0.000 deg,	P = 30.000 deg,	R = 139.825 deg
};
P[122]{
   GP1:
	UF : 0, UT : 1,		CONFIG : 'N U T, 0, 0, 0',
	X = 1226.351  mm,	Y = -183.148  mm,	Z = -239.482  mm,
	W = 0.000 deg,	P = 30.000 deg,	R = 139.825 deg
};
P[123]{
   GP1:
	UF : 0, UT : 1,		CONFIG : 'N U T, 0, 0, 0',
	X = 1227.631  mm,	Y = -181.632  mm,	Z = -239.732  mm,
	W = 0.000 deg,	P = 30.000 deg,	R = 139.825 deg
};
P[124]{
   GP1:
	UF : 0, UT : 1,		CONFIG : 'N U T, 0, 0, 0',
	X = 1228.911  mm,	Y = -180.116  mm,	Z = -239.982  mm,
	W = 0.000 deg,	P = 30.000 deg,	R = 139.825 deg
};
P[125]{
   GP1:
	UF : 0, UT : 1,		CONFIG : 'N U T, 0, 0, 0',
	X = 1230.191  mm,	Y = -178.599  mm,	Z = -240.232  mm,
	W = 0.000 deg,	P = 30.000 deg,	R = 139.825 deg
};
P[126]{
   GP1:
	UF : 0, UT : 1,		CONFIG : 'N U T, 0, 0, 0',
	X = 1231.471  mm,	Y = -177.083  mm,	Z = -240.481  mm,
	W = 0.000 deg,	P = 30.000 deg,	R = 139.825 deg
};
P[127]{
   GP1:
	UF : 0, UT : 1,		CONFIG : 'N U T, 0, 0, 0',
	X = 1232.751  mm,	Y = -175.567  mm,	Z = -240.731  mm,
	W = 0.000 deg,	P = 30.000 deg,	R = 139.825 deg
};
P[128]{
   GP1:
	UF : 0, UT : 1,		CONFIG : 'N U T, 0, 0, 0',
	X = 1234.032  mm,	Y = -174.051  mm,	Z = -240.981  mm,
	W = 0.000 deg,	P = 30.000 deg,	R = 139.825 deg
};
P[129]{
   GP1:
	UF : 0, UT : 1,		CONFIG : 'N U T, 0, 0, 0',
	X = 1235.312  mm,	Y = -172.535  mm,	Z = -241.231  mm,
	W = 0.000 deg,	P = 30.000 deg,	R = 139.825 deg
};
P[130]{
   GP1:
	UF : 0, UT : 1,		CONFIG : 'N U T, 0, 0, 0',
	X = 1236.592  mm,	Y = -171.019  mm,	Z = -241.481  mm,
	W = 0.000 deg,	P = 30.000 deg,	R = 139.825 deg
};
P[131]{
   GP1:
	UF : 0, UT : 1,		CONFIG : 'N U T, 0, 0, 0',
	X = 1237.872  mm,	Y = -169.502  mm,	Z = -241.731  mm,
	W = 0.000 deg,	P = 30.000 deg,	R = 139.825 deg
};
P[132]{
   GP1:
	UF : 0, UT : 1,		CONFIG : 'N U T, 0, 0, 0',
	X = 1239.152  mm,	Y = -167.986  mm,	Z = -241.981  mm,
	W = 0.000 deg,	P = 30.000 deg,	R = 139.825 deg
};
P[133]{
   GP1:
	UF : 0, UT : 1,		CONFIG : 'N U T, 0, 0, 0',
	X = 1240.432  mm,	Y = -166.470  mm,	Z = -242.231  mm,
	W = 0.000 deg,	P = 30.000 deg,	R = 139.825 deg
};
P[134]{
   GP1:
	UF : 0, UT : 1,		CONFIG : 'N U T, 0, 0, 0',
	X = 1241.712  mm,	Y = -164.954  mm,	Z = -242.480  mm,
	W = 0.000 deg,	P = 30.000 deg,	R = 141.055 deg
};
P[135]{
   GP1:
	UF : 0, UT : 1,		CONFIG : 'N U T, 0, 0, 0',
	X = 1242.993  mm,	Y = -163.438  mm,	Z = -242.730  mm,
	W = 0.000 deg,	P = 30.000 deg,	R = 149.779 deg
};
P[136]{
   GP1:
	UF : 0, UT : 1,		CONFIG : 'N U T, 0, 0, 0',
	X = 1244.273  mm,	Y = -161.921  mm,	Z = -242.980  mm,
	W = 0.000 deg,	P = 30.000 deg,	R = 158.503 deg
};
P[137]{
   GP1:
	UF : 0, UT : 1,		CONFIG : 'N U T, 0, 0, 0',
	X = 1245.553  mm,	Y = -160.405  mm,	Z = -243.230  mm,
	W = 0.000 deg,	P = 30.000 deg,	R = 167.226 deg
};
P[138]{
   GP1:
	UF : 0, UT : 1,		CONFIG : 'N U T, 0, 0, 0',
	X = 1246.833  mm,	Y = -158.889  mm,	Z = -243.480  mm,
	W = 0.000 deg,	P = 30.000 deg,	R = 175.950 deg
};
P[139]{
   GP1:
	UF : 0, UT : 1,		CONFIG : 'N U T, 0, 0, 0',
	X = 1248.113  mm,	Y = -157.373  mm,	Z = -243.730  mm,
	W = 0.000 deg,	P = 30.000 deg,	R = -176.557 deg
};
P[140]{
   GP1:
	UF : 0, UT : 1,		CONFIG : 'N U T, 0, 0, 0',
	X = 1245.929  mm,	Y = -163.288  mm,	Z = -243.763  mm,
	W = 0.000 deg,	P = 30.000 deg,	R = -176.557 deg
};
P[141]{
   GP1:
	UF : 0, UT : 1,		CONFIG : 'N U T, 0, 0, 0',
	X = 1245.837  mm,	Y = -162.492  mm,	Z = -243.720  mm,
	W = 0.000 deg,	P = 30.000 deg,	R = -176.557 deg
};
P[142]{
   GP1:
	UF : 0, UT : 1,		CONFIG : 'N U T, 0, 0, 0',
	X = 1245.717  mm,	Y = -160.496  mm,	Z = -243.670  mm,
	W = 0.000 deg,	P = 30.000 deg,	R = -176.557 deg
};
P[143]{
   GP1:
	UF : 0, UT : 1,		CONFIG : 'N U T, 0, 0, 0',
	X = 1245.597  mm,	Y = -158.501  mm,	Z = -243.621  mm,
	W = 0.000 deg,	P = 30.000 deg,	R = -176.557 deg
};
P[144]{
   GP1:
	UF : 0, UT : 1,		CONFIG : 'N U T, 0, 0, 0',
	X = 1245.477  mm,	Y = -156.505  mm,	Z = -243.571  mm,
	W = 0.000 deg,	P = 30.000 deg,	R = -176.557 deg
};
P[145]{
   GP1:
	UF : 0, UT : 1,		CONFIG : 'N U T, 0, 0, 0',
	X = 1245.357  mm,	Y = -154.509  mm,	Z = -243.522  mm,
	W = 0.000 deg,	P = 30.000 deg,	R = -176.557 deg
};
P[146]{
   GP1:
	UF : 0, UT : 1,		CONFIG : 'N U T, 0, 0, 0',
	X = 1245.237  mm,	Y = -152.513  mm,	Z = -243.472  mm,
	W = 0.000 deg,	P = 30.000 deg,	R = -176.557 deg
};
P[147]{
   GP1:
	UF : 0, UT : 1,		CONFIG : 'N U T, 0, 0, 0',
	X = 1245.117  mm,	Y = -150.518  mm,	Z = -243.422  mm,
	W = 0.000 deg,	P = 30.000 deg,	R = -176.557 deg
};
P[148]{
   GP1:
	UF : 0, UT : 1,		CONFIG : 'N U T, 0, 0, 0',
	X = 1244.997  mm,	Y = -148.522  mm,	Z = -243.373  mm,
	W = 0.000 deg,	P = 30.000 deg,	R = -176.557 deg
};
P[149]{
   GP1:
	UF : 0, UT : 1,		CONFIG : 'N U T, 0, 0, 0',
	X = 1244.876  mm,	Y = -146.526  mm,	Z = -243.323  mm,
	W = 0.000 deg,	P = 30.000 deg,	R = -176.557 deg
};
P[150]{
   GP1:
	UF : 0, UT : 1,		CONFIG : 'N U T, 0, 0, 0',
	X = 1244.756  mm,	Y = -144.530  mm,	Z = -243.274  mm,
	W = 0.000 deg,	P = 30.000 deg,	R = -176.557 deg
};
P[151]{
   GP1:
	UF : 0, UT : 1,		CONFIG : 'N U T, 0, 0, 0',
	X = 1244.636  mm,	Y = -142.534  mm,	Z = -243.224  mm,
	W = 0.000 deg,	P = 30.000 deg,	R = -176.557 deg
};
P[152]{
   GP1:
	UF : 0, UT : 1,		CONFIG : 'N U T, 0, 0, 0',
	X = 1244.516  mm,	Y = -140.539  mm,	Z = -243.175  mm,
	W = 0.000 deg,	P = 30.000 deg,	R = -176.557 deg
};
P[153]{
   GP1:
	UF : 0, UT : 1,		CONFIG : 'N U T, 0, 0, 0',
	X = 1244.396  mm,	Y = -138.543  mm,	Z = -243.125  mm,
	W = 0.000 deg,	P = 30.000 deg,	R = -176.557 deg
};
P[154]{
   GP1:
	UF : 0, UT : 1,		CONFIG : 'N U T, 0, 0, 0',
	X = 1244.276  mm,	Y = -136.547  mm,	Z = -243.076  mm,
	W = 0.000 deg,	P = 30.000 deg,	R = -176.557 deg
};
P[155]{
   GP1:
	UF : 0, UT : 1,		CONFIG : 'N U T, 0, 0, 0',
	X = 1244.156  mm,	Y = -134.551  mm,	Z = -243.026  mm,
	W = 0.000 deg,	P = 30.000 deg,	R = -176.557 deg
};
P[156]{
   GP1:
	UF : 0, UT : 1,		CONFIG : 'N U T, 0, 0, 0',
	X = 1244.036  mm,	Y = -132.556  mm,	Z = -242.976  mm,
	W = 0.000 deg,	P = 30.000 deg,	R = -176.557 deg
};
P[157]{
   GP1:
	UF : 0, UT : 1,		CONFIG : 'N U T, 0, 0, 0',
	X = 1243.916  mm,	Y = -130.560  mm,	Z = -242.927  mm,
	W = 0.000 deg,	P = 30.000 deg,	R = -176.557 deg
};
P[158]{
   GP1:
	UF : 0, UT : 1,		CONFIG : 'N U T, 0, 0, 0',
	X = 1243.796  mm,	Y = -128.564  mm,	Z = -242.877  mm,
	W = 0.000 deg,	P = 30.000 deg,	R = -176.557 deg
};
P[159]{
   GP1:
	UF : 0, UT : 1,		CONFIG : 'N U T, 0, 0, 0',
	X = 1243.676  mm,	Y = -126.568  mm,	Z = -242.828  mm,
	W = 0.000 deg,	P = 30.000 deg,	R = -176.557 deg
};
P[160]{
   GP1:
	UF : 0, UT : 1,		CONFIG : 'N U T, 0, 0, 0',
	X = 1243.556  mm,	Y = -124.572  mm,	Z = -242.778  mm,
	W = 0.000 deg,	P = 30.000 deg,	R = -176.557 deg
};
P[161]{
   GP1:
	UF : 0, UT : 1,		CONFIG : 'N U T, 0, 0, 0',
	X = 1243.436  mm,	Y = -122.577  mm,	Z = -242.729  mm,
	W = 0.000 deg,	P = 30.000 deg,	R = -176.557 deg
};
P[162]{
   GP1:
	UF : 0, UT : 1,		CONFIG : 'N U T, 0, 0, 0',
	X = 1243.316  mm,	Y = -120.581  mm,	Z = -242.679  mm,
	W = 0.000 deg,	P = 30.000 deg,	R = -176.557 deg
};
P[163]{
   GP1:
	UF : 0, UT : 1,		CONFIG : 'N U T, 0, 0, 0',
	X = 1243.196  mm,	Y = -118.585  mm,	Z = -242.630  mm,
	W = 0.000 deg,	P = 30.000 deg,	R = -176.557 deg
};
P[164]{
   GP1:
	UF : 0, UT : 1,		CONFIG : 'N U T, 0, 0, 0',
	X = 1243.076  mm,	Y = -116.589  mm,	Z = -242.580  mm,
	W = 0.000 deg,	P = 30.000 deg,	R = -169.254 deg
};
P[165]{
   GP1:
	UF : 0, UT : 1,		CONFIG : 'N U T, 0, 0, 0',
	X = 1242.956  mm,	Y = -114.594  mm,	Z = -242.530  mm,
	W = 0.000 deg,	P = 30.000 deg,	R = -160.840 deg
};
P[166]{
   GP1:
	UF : 0, UT : 1,		CONFIG : 'N U T, 0, 0, 0',
	X = 1242.835  mm,	Y = -112.598  mm,	Z = -242.481  mm,
	W = 0.000 deg,	P = 30.000 deg,	R = -152.425 deg
};
P[167]{
   GP1:
	UF : 0, UT : 1,		CONFIG : 'N U T, 0, 0, 0',
	X = 1242.715  mm,	Y = -110.602  mm,	Z = -242.431  mm,
	W = 0.000 deg,	P = 30.000 deg,	R = -144.010 deg
};
P[168]{
   GP1:
	UF : 0, UT : 1,		CONFIG : 'N U T, 0, 0, 0',
	X = 1242.595  mm,	Y = -108.606  mm,	Z = -242.382  mm,
	W = 0.000 deg,	P = 30.000 deg,	R = -135.595 deg
};
P[169]{
   GP1:
	UF : 0, UT : 1,		CONFIG : 'N U T, 0, 0, 0',
	X = 1244.490  mm,	Y = -113.472  mm,	Z = -242.371  mm,
	W = 0.000 deg,	P = 30.000 deg,	R = -134.483 deg
};
P[170]{
   GP1:
	UF : 0, UT : 1,		CONFIG : 'N U T, 0, 0, 0',
	X = 1244.451  mm,	Y = -113.616  mm,	Z = -242.141  mm,
	W = 0.000 deg,	P = 30.000 deg,	R = -134.483 deg
};
P[171]{
   GP1:
	UF : 0, UT : 1,		CONFIG : 'N U T, 0, 0, 0',
	X = 1243.040  mm,	Y = -112.230  mm,	Z = -241.845  mm,
	W = 0.000 deg,	P = 30.000 deg,	R = -134.483 deg
};
P[172]{
   GP1:
	UF : 0, UT : 1,		CONFIG : 'N U T, 0, 0, 0',
	X = 1241.629  mm,	Y = -110.845  mm,	Z = -241.548  mm,
	W = 0.000 deg,	P = 30.000 deg,	R = -134.483 deg
};
P[173]{
   GP1:
	UF : 0, UT : 1,		CONFIG : 'N U T, 0, 0, 0',
	X = 1240.218  mm,	Y = -109.459  mm,	Z = -241.252  mm,
	W = 0.000 deg,	P = 30.000 deg,	R = -134.483 deg
};
P[174]{
   GP1:
	UF : 0, UT : 1,		CONFIG : 'N U T, 0, 0, 0',
	X = 1238.807  mm,	Y = -108.073  mm,	Z = -240.955  mm,
	W = 0.000 deg,	P = 30.000 deg,	R = -134.483 deg
};
P[175]{
   GP1:
	UF : 0, UT : 1,		CONFIG : 'N U T, 0, 0, 0',
	X = 1237.396  mm,	Y = -106.687  mm,	Z = -240.659  mm,
	W = 0.000 deg,	P = 30.000 deg,	R = -134.483 deg
};
P[176]{
   GP1:
	UF : 0, UT : 1,		CONFIG : 'N U T, 0, 0, 0',
	X = 1235.985  mm,	Y = -105.301  mm,	Z = -240.362  mm,
	W = 0.000 deg,	P = 30.000 deg,	R = -134.483 deg
};
P[177]{
   GP1:
	UF : 0, UT : 1,		CONFIG : 'N U T, 0, 0, 0',
	X = 1234.573  mm,	Y = -103.915  mm,	Z = -240.066  mm,
	W = 0.000 deg,	P = 30.000 deg,	R = -134.483 deg
};
P[178]{
   GP1:
	UF : 0, UT : 1,		CONFIG : 'N U T, 0, 0, 0',
	X = 1233.162  mm,	Y = -102.529  mm,	Z = -239.769  mm,
	W = 0.000 deg,	P = 30.000 deg,	R = -134.483 deg
};
P[179]{
   GP1:
	UF : 0, UT : 1,		CONFIG : 'N U T, 0, 0, 0',
	X = 1231.751  mm,	Y = -101.143  mm,	Z = -239.473  mm,
	W = 0.000 deg,	P = 30.000 deg,	R = -134.483 deg
};
P[180]{
   GP1:
	UF : 0, UT : 1,		CONFIG : 'N U T, 0, 0, 0',
	X = 1230.340  mm,	Y = -99.757  mm,	Z = -239.176  mm,
	W = 0.000 deg,	P = 30.000 deg,	R = -134.483 deg
};
P[181]{
   GP1:
	UF : 0, UT : 1,		CONFIG : 'N U T, 0, 0, 0',
	X = 1228.929  mm,	Y = -98.371  mm,	Z = -238.880  mm,
	W = 0.000 deg,	P = 30.000 deg,	R = -134.483 deg
};
P[182]{
   GP1:
	UF : 0, UT : 1,		CONFIG : 'N U T, 0, 0, 0',
	X = 1227.518  mm,	Y = -96.985  mm,	Z = -238.583  mm,
	W = 0.000 deg,	P = 30.000 deg,	R = -134.483 deg
};
P[183]{
   GP1:
	UF : 0, UT : 1,		CONFIG : 'N U T, 0, 0, 0',
	X = 1226.107  mm,	Y = -95.600  mm,	Z = -238.287  mm,
	W = 0.000 deg,	P = 30.000 deg,	R = -134.483 deg
};
P[184]{
   GP1:
	UF : 0, UT : 1,		CONFIG : 'N U T, 0, 0, 0',
	X = 1224.695  mm,	Y = -94.214  mm,	Z = -237.990  mm,
	W = 0.000 deg,	P = 30.000 deg,	R = -134.483 deg
};
P[185]{
   GP1:
	UF : 0, UT : 1,		CONFIG : 'N U T, 0, 0, 0',
	X = 1223.284  mm,	Y = -92.828  mm,	Z = -237.694  mm,
	W = 0.000 deg,	P = 30.000 deg,	R = -134.483 deg
};
P[186]{
   GP1:
	UF : 0, UT : 1,		CONFIG : 'N U T, 0, 0, 0',
	X = 1221.873  mm,	Y = -91.442  mm,	Z = -237.397  mm,
	W = 0.000 deg,	P = 30.000 deg,	R = -134.483 deg
};
P[187]{
   GP1:
	UF : 0, UT : 1,		CONFIG : 'N U T, 0, 0, 0',
	X = 1220.462  mm,	Y = -90.056  mm,	Z = -237.101  mm,
	W = 0.000 deg,	P = 30.000 deg,	R = -134.483 deg
};
P[188]{
   GP1:
	UF : 0, UT : 1,		CONFIG : 'N U T, 0, 0, 0',
	X = 1219.051  mm,	Y = -88.670  mm,	Z = -236.804  mm,
	W = 0.000 deg,	P = 30.000 deg,	R = -134.483 deg
};
P[189]{
   GP1:
	UF : 0, UT : 1,		CONFIG : 'N U T, 0, 0, 0',
	X = 1217.640  mm,	Y = -87.284  mm,	Z = -236.508  mm,
	W = 0.000 deg,	P = 30.000 deg,	R = -134.483 deg
};
P[190]{
   GP1:
	UF : 0, UT : 1,		CONFIG : 'N U T, 0, 0, 0',
	X = 1216.229  mm,	Y = -85.898  mm,	Z = -236.211  mm,
	W = 0.000 deg,	P = 30.000 deg,	R = -141.380 deg
};
P[191]{
   GP1:
	UF : 0, UT : 1,		CONFIG : 'N U T, 0, 0, 0',
	X = 1214.817  mm,	Y = -84.512  mm,	Z = -235.915  mm,
	W = 0.000 deg,	P = 30.000 deg,	R = -150.295 deg
};
P[192]{
   GP1:
	UF : 0, UT : 1,		CONFIG : 'N U T, 0, 0, 0',
	X = 1213.406  mm,	Y = -83.126  mm,	Z = -235.618  mm,
	W = 0.000 deg,	P = 30.000 deg,	R = -159.209 deg
};
P[193]{
   GP1:
	UF : 0, UT : 1,		CONFIG : 'N U T, 0, 0, 0',
	X = 1211.995  mm,	Y = -81.740  mm,	Z = -235.321  mm,
	W = 0.000 deg,	P = 30.000 deg,	R = -168.124 deg
};
P[194]{
   GP1:
	UF : 0, UT : 1,		CONFIG : 'N U T, 0, 0, 0',
	X = 1210.584  mm,	Y = -80.355  mm,	Z = -235.025  mm,
	W = 0.000 deg,	P = 30.000 deg,	R = -177.038 deg
};
P[195]{
   GP1:
	UF : 0, UT : 1,		CONFIG : 'N U T, 0, 0, 0',
	X = 1209.173  mm,	Y = -78.969  mm,	Z = -234.728  mm,
	W = 0.000 deg,	P = 30.000 deg,	R = -179.056 deg
};
P[196]{
   GP1:
	UF : 0, UT : 1,		CONFIG : 'N U T, 0, 0, 0',
	X = 1206.063  mm,	Y = -72.688  mm,	Z = -234.693  mm,
	W = 0.000 deg,	P = 30.000 deg,	R = -179.056 deg
};
P[197]{
   GP1:
	UF : 0, UT : 1,		CONFIG : 'N U T, 0, 0, 0',
	X = 1205.984  mm,	Y = -70.072  mm,	Z = -234.671  mm,
	W = 0.000 deg,	P = 30.000 deg,	R = -179.056 deg
};
P[198]{
   GP1:
	UF : 0, UT : 1,		CONFIG : 'N U T, 0, 0, 0',
	X = 1205.951  mm,	Y = -68.073  mm,	Z = -234.647  mm,
	W = 0.000 deg,	P = 30.000 deg,	R = -179.056 deg
};
P[199]{
   GP1:
	UF : 0, UT : 1,		CONFIG : 'N U T, 0, 0, 0',
	X = 1205.918  mm,	Y = -66.073  mm,	Z = -234.622  mm,
	W = 0.000 deg,	P = 30.000 deg,	R = -179.056 deg
};
P[200]{
   GP1:
	UF : 0, UT : 1,		CONFIG : 'N U T, 0, 0, 0',
	X = 1205.885  mm,	Y = -64.074  mm,	Z = -234.597  mm,
	W = 0.000 deg,	P = 30.000 deg,	R = -179.056 deg
};
P[201]{
   GP1:
	UF : 0, UT : 1,		CONFIG : 'N U T, 0, 0, 0',
	X = 1205.852  mm,	Y = -62.074  mm,	Z = -234.572  mm,
	W = 0.000 deg,	P = 30.000 deg,	R = -179.056 deg
};
P[202]{
   GP1:
	UF : 0, UT : 1,		CONFIG : 'N U T, 0, 0, 0',
	X = 1205.819  mm,	Y = -60.075  mm,	Z = -234.547  mm,
	W = 0.000 deg,	P = 30.000 deg,	R = -179.056 deg
};
P[203]{
   GP1:
	UF : 0, UT : 1,		CONFIG : 'N U T, 0, 0, 0',
	X = 1205.786  mm,	Y = -58.075  mm,	Z = -234.523  mm,
	W = 0.000 deg,	P = 30.000 deg,	R = -179.056 deg
};
P[204]{
   GP1:
	UF : 0, UT : 1,		CONFIG : 'N U T, 0, 0, 0',
	X = 1205.753  mm,	Y = -56.075  mm,	Z = -234.498  mm,
	W = 0.000 deg,	P = 30.000 deg,	R = -179.056 deg
};
P[205]{
   GP1:
	UF : 0, UT : 1,		CONFIG : 'N U T, 0, 0, 0',
	X = 1205.720  mm,	Y = -54.076  mm,	Z = -234.473  mm,
	W = 0.000 deg,	P = 30.000 deg,	R = -179.056 deg
};
P[206]{
   GP1:
	UF : 0, UT : 1,		CONFIG : 'N U T, 0, 0, 0',
	X = 1205.687  mm,	Y = -52.076  mm,	Z = -234.448  mm,
	W = 0.000 deg,	P = 30.000 deg,	R = -179.056 deg
};
P[207]{
   GP1:
	UF : 0, UT : 1,		CONFIG : 'N U T, 0, 0, 0',
	X = 1205.654  mm,	Y = -50.077  mm,	Z = -234.424  mm,
	W = 0.000 deg,	P = 30.000 deg,	R = -179.056 deg
};
P[208]{
   GP1:
	UF : 0, UT : 1,		CONFIG : 'N U T, 0, 0, 0',
	X = 1205.621  mm,	Y = -48.077  mm,	Z = -234.399  mm,
	W = 0.000 deg,	P = 30.000 deg,	R = -179.056 deg
};
P[209]{
   GP1:
	UF : 0, UT : 1,		CONFIG : 'N U T, 0, 0, 0',
	X = 1205.588  mm,	Y = -46.078  mm,	Z = -234.374  mm,
	W = 0.000 deg,	P = 30.000 deg,	R = -179.056 deg
};
P[210]{
   GP1:
	UF : 0, UT : 1,		CONFIG : 'N U T, 0, 0, 0',
	X = 1205.555  mm,	Y = -44.078  mm,	Z = -234.349  mm,
	W = 0.000 deg,	P = 30.000 deg,	R = -179.056 deg
};
P[211]{
   GP1:
	UF : 0, UT : 1,		CONFIG : 'N U T, 0, 0, 0',
	X = 1205.522  mm,	Y = -42.078  mm,	Z = -234.325  mm,
	W = 0.000 deg,	P = 30.000 deg,	R = -179.056 deg
};
P[212]{
   GP1:
	UF : 0, UT : 1,		CONFIG : 'N U T, 0, 0, 0',
	X = 1205.489  mm,	Y = -40.079  mm,	Z = -234.300  mm,
	W = 0.000 deg,	P = 30.000 deg,	R = -179.056 deg
};
P[213]{
   GP1:
	UF : 0, UT : 1,		CONFIG : 'N U T, 0, 0, 0',
	X = 1205.456  mm,	Y = -38.079  mm,	Z = -234.275  mm,
	W = 0.000 deg,	P = 30.000 deg,	R = -179.056 deg
};
P[214]{
   GP1:
	UF : 0, UT : 1,		CONFIG : 'N U T, 0, 0, 0',
	X = 1205.423  mm,	Y = -36.080  mm,	Z = -234.250  mm,
	W = 0.000 deg,	P = 30.000 deg,	R = -179.056 deg
};
P[215]{
   GP1:
	UF : 0, UT : 1,		CONFIG : 'N U T, 0, 0, 0',
	X = 1205.391  mm,	Y = -34.080  mm,	Z = -234.226  mm,
	W = 0.000 deg,	P = 30.000 deg,	R = -179.056 deg
};
P[216]{
   GP1:
	UF : 0, UT : 1,		CONFIG : 'N U T, 0, 0, 0',
	X = 1205.358  mm,	Y = -32.081  mm,	Z = -234.201  mm,
	W = 0.000 deg,	P = 30.000 deg,	R = -179.056 deg
};
P[217]{
   GP1:
	UF : 0, UT : 1,		CONFIG : 'N U T, 0, 0, 0',
	X = 1205.325  mm,	Y = -30.081  mm,	Z = -234.176  mm,
	W = 0.000 deg,	P = 30.000 deg,	R = -179.056 deg
};
P[218]{
   GP1:
	UF : 0, UT : 1,		CONFIG : 'N U T, 0, 0, 0',
	X = 1205.292  mm,	Y = -28.081  mm,	Z = -234.151  mm,
	W = 0.000 deg,	P = 30.000 deg,	R = -179.056 deg
};
P[219]{
   GP1:
	UF : 0, UT : 1,		CONFIG : 'N U T, 0, 0, 0',
	X = 1205.259  mm,	Y = -26.082  mm,	Z = -234.126  mm,
	W = 0.000 deg,	P = 30.000 deg,	R = -179.056 deg
};
P[220]{
   GP1:
	UF : 0, UT : 1,		CONFIG : 'N U T, 0, 0, 0',
	X = 1205.226  mm,	Y = -24.082  mm,	Z = -234.102  mm,
	W = 0.000 deg,	P = 30.000 deg,	R = -179.056 deg
};
P[221]{
   GP1:
	UF : 0, UT : 1,		CONFIG : 'N U T, 0, 0, 0',
	X = 1205.193  mm,	Y = -22.083  mm,	Z = -234.077  mm,
	W = 0.000 deg,	P = 30.000 deg,	R = -179.056 deg
};
P[222]{
   GP1:
	UF : 0, UT : 1,		CONFIG : 'N U T, 0, 0, 0',
	X = 1205.160  mm,	Y = -20.083  mm,	Z = -234.052  mm,
	W = 0.000 deg,	P = 30.000 deg,	R = 164.852 deg
};
P[223]{
   GP1:
	UF : 0, UT : 1,		CONFIG : 'N U T, 0, 0, 0',
	X = 1205.127  mm,	Y = -18.084  mm,	Z = -234.027  mm,
	W = 0.000 deg,	P = 30.000 deg,	R = 156.296 deg
};
P[224]{
   GP1:
	UF : 0, UT : 1,		CONFIG : 'N U T, 0, 0, 0',
	X = 1205.094  mm,	Y = -16.084  mm,	Z = -234.003  mm,
	W = 0.000 deg,	P = 30.000 deg,	R = 147.739 deg
};
P[225]{
   GP1:
	UF : 0, UT : 1,		CONFIG : 'N U T, 0, 0, 0',
	X = 1205.061  mm,	Y = -14.084  mm,	Z = -233.978  mm,
	W = 0.000 deg,	P = 30.000 deg,	R = 139.183 deg
};
P[226]{
   GP1:
	UF : 0, UT : 1,		CONFIG : 'N U T, 0, 0, 0',
	X = 1205.195  mm,	Y = -10.687  mm,	Z = -233.960  mm,
	W = 0.000 deg,	P = 30.000 deg,	R = 138.161 deg
};
P[227]{
   GP1:
	UF : 0, UT : 1,		CONFIG : 'N U T, 0, 0, 0',
	X = 1207.945  mm,	Y = -5.392  mm,	Z = -234.038  mm,
	W = 0.000 deg,	P = 30.000 deg,	R = 138.161 deg
};
P[228]{
   GP1:
	UF : 0, UT : 1,		CONFIG : 'N U T, 0, 0, 0',
	X = 1209.265  mm,	Y = -3.918  mm,	Z = -234.324  mm,
	W = 0.000 deg,	P = 30.000 deg,	R = 138.161 deg
};
P[229]{
   GP1:
	UF : 0, UT : 1,		CONFIG : 'N U T, 0, 0, 0',
	X = 1210.585  mm,	Y = -2.443  mm,	Z = -234.610  mm,
	W = 0.000 deg,	P = 30.000 deg,	R = 138.161 deg
};
P[230]{
   GP1:
	UF : 0, UT : 1,		CONFIG : 'N U T, 0, 0, 0',
	X = 1211.906  mm,	Y = -0.968  mm,	Z = -234.896  mm,
	W = 0.000 deg,	P = 30.000 deg,	R = 138.161 deg
};
P[231]{
   GP1:
	UF : 0, UT : 1,		CONFIG : 'N U T, 0, 0, 0',
	X = 1213.226  mm,	Y = 0.506  mm,	Z = -235.181  mm,
	W = 0.000 deg,	P = 30.000 deg,	R = 138.161 deg
};
P[232]{
   GP1:
	UF : 0, UT : 1,		CONFIG : 'N U T, 0, 0, 0',
	X = 1214.547  mm,	Y = 1.981  mm,	Z = -235.467  mm,
	W = 0.000 deg,	P = 30.000 deg,	R = 138.161 deg
};
P[233]{
   GP1:
	UF : 0, UT : 1,		CONFIG : 'N U T, 0, 0, 0',
	X = 1215.867  mm,	Y = 3.456  mm,	Z = -235.753  mm,
	W = 0.000 deg,	P = 30.000 deg,	R = 138.161 deg
};
P[234]{
   GP1:
	UF : 0, UT : 1,		CONFIG : 'N U T, 0, 0, 0',
	X = 1217.187  mm,	Y = 4.931  mm,	Z = -236.039  mm,
	W = 0.000 deg,	P = 30.000 deg,	R = 138.161 deg
};
P[235]{
   GP1:
	UF : 0, UT : 1,		CONFIG : 'N U T, 0, 0, 0',
	X = 1218.508  mm,	Y = 6.405  mm,	Z = -236.325  mm,
	W = 0.000 deg,	P = 30.000 deg,	R = 138.161 deg
};
P[236]{
   GP1:
	UF : 0, UT : 1,		CONFIG : 'N U T, 0, 0, 0',
	X = 1219.828  mm,	Y = 7.880  mm,	Z = -236.611  mm,
	W = 0.000 deg,	P = 30.000 deg,	R = 138.161 deg
};
P[237]{
   GP1:
	UF : 0, UT : 1,		CONFIG : 'N U T, 0, 0, 0',
	X = 1221.148  mm,	Y = 9.355  mm,	Z = -236.897  mm,
	W = 0.000 deg,	P = 30.000 deg,	R = 138.161 deg
};
P[238]{
   GP1:
	UF : 0, UT : 1,		CONFIG : 'N U T, 0, 0, 0',
	X = 1222.469  mm,	Y = 10.830  mm,	Z = -237.183  mm,
	W = 0.000 deg,	P = 30.000 deg,	R = 138.161 deg
};
P[239]{
   GP1:
	UF : 0, UT : 1,		CONFIG : 'N U T, 0, 0, 0',
	X = 1223.789  mm,	Y = 12.304  mm,	Z = -237.469  mm,
	W = 0.000 deg,	P = 30.000 deg,	R = 138.161 deg
};
P[240]{
   GP1:
	UF : 0, UT : 1,		CONFIG : 'N U T, 0, 0, 0',
	X = 1225.110  mm,	Y = 13.779  mm,	Z = -237.755  mm,
	W = 0.000 deg,	P = 30.000 deg,	R = 138.161 deg
};
P[241]{
   GP1:
	UF : 0, UT : 1,		CONFIG : 'N U T, 0, 0, 0',
	X = 1226.430  mm,	Y = 15.254  mm,	Z = -238.041  mm,
	W = 0.000 deg,	P = 30.000 deg,	R = 138.161 deg
};
P[242]{
   GP1:
	UF : 0, UT : 1,		CONFIG : 'N U T, 0, 0, 0',
	X = 1227.750  mm,	Y = 16.729  mm,	Z = -238.327  mm,
	W = 0.000 deg,	P = 30.000 deg,	R = 138.161 deg
};
P[243]{
   GP1:
	UF : 0, UT : 1,		CONFIG : 'N U T, 0, 0, 0',
	X = 1229.071  mm,	Y = 18.203  mm,	Z = -238.613  mm,
	W = 0.000 deg,	P = 30.000 deg,	R = 138.161 deg
};
P[244]{
   GP1:
	UF : 0, UT : 1,		CONFIG : 'N U T, 0, 0, 0',
	X = 1230.391  mm,	Y = 19.678  mm,	Z = -238.899  mm,
	W = 0.000 deg,	P = 30.000 deg,	R = 138.161 deg
};
P[245]{
   GP1:
	UF : 0, UT : 1,		CONFIG : 'N U T, 0, 0, 0',
	X = 1231.711  mm,	Y = 21.153  mm,	Z = -239.185  mm,
	W = 0.000 deg,	P = 30.000 deg,	R = 138.161 deg
};
P[246]{
   GP1:
	UF : 0, UT : 1,		CONFIG : 'N U T, 0, 0, 0',
	X = 1233.032  mm,	Y = 22.628  mm,	Z = -239.471  mm,
	W = 0.000 deg,	P = 30.000 deg,	R = 140.626 deg
};
P[247]{
   GP1:
	UF : 0, UT : 1,		CONFIG : 'N U T, 0, 0, 0',
	X = 1234.352  mm,	Y = 24.102  mm,	Z = -239.756  mm,
	W = 0.000 deg,	P = 30.000 deg,	R = 149.685 deg
};
P[248]{
   GP1:
	UF : 0, UT : 1,		CONFIG : 'N U T, 0, 0, 0',
	X = 1235.673  mm,	Y = 25.577  mm,	Z = -240.042  mm,
	W = 0.000 deg,	P = 30.000 deg,	R = 158.745 deg
};
P[249]{
   GP1:
	UF : 0, UT : 1,		CONFIG : 'N U T, 0, 0, 0',
	X = 1236.993  mm,	Y = 27.052  mm,	Z = -240.328  mm,
	W = 0.000 deg,	P = 30.000 deg,	R = 167.804 deg
};
P[250]{
   GP1:
	UF : 0, UT : 1,		CONFIG : 'N U T, 0, 0, 0',
	X = 1238.313  mm,	Y = 28.527  mm,	Z = -240.614  mm,
	W = 0.000 deg,	P = 30.000 deg,	R = 176.864 deg
};
P[251]{
   GP1:
	UF : 0, UT : 1,		CONFIG : 'N U T, 0, 0, 0',
	X = 1239.634  mm,	Y = 30.001  mm,	Z = -240.900  mm,
	W = 0.000 deg,	P = 30.000 deg,	R = -176.541 deg
};
P[252]{
   GP1:
	UF : 0, UT : 1,		CONFIG : 'N U T, 0, 0, 0',
	X = 1239.075  mm,	Y = 28.891  mm,	Z = -241.092  mm,
	W = 0.000 deg,	P = 30.000 deg,	R = -176.541 deg
};
P[253]{
   GP1:
	UF : 0, UT : 1,		CONFIG : 'N U T, 0, 0, 0',
	X = 1237.948  mm,	Y = 24.374  mm,	Z = -241.081  mm,
	W = 0.000 deg,	P = 30.000 deg,	R = -176.541 deg
};
P[254]{
   GP1:
	UF : 0, UT : 1,		CONFIG : 'N U T, 0, 0, 0',
	X = 1237.828  mm,	Y = 26.370  mm,	Z = -241.048  mm,
	W = 0.000 deg,	P = 30.000 deg,	R = -176.541 deg
};
P[255]{
   GP1:
	UF : 0, UT : 1,		CONFIG : 'N U T, 0, 0, 0',
	X = 1237.707  mm,	Y = 28.366  mm,	Z = -241.016  mm,
	W = 0.000 deg,	P = 30.000 deg,	R = -176.541 deg
};
P[256]{
   GP1:
	UF : 0, UT : 1,		CONFIG : 'N U T, 0, 0, 0',
	X = 1237.586  mm,	Y = 30.362  mm,	Z = -240.983  mm,
	W = 0.000 deg,	P = 30.000 deg,	R = -176.541 deg
};
P[257]{
   GP1:
	UF : 0, UT : 1,		CONFIG : 'N U T, 0, 0, 0',
	X = 1237.466  mm,	Y = 32.358  mm,	Z = -240.950  mm,
	W = 0.000 deg,	P = 30.000 deg,	R = -176.541 deg
};
P[258]{
   GP1:
	UF : 0, UT : 1,		CONFIG : 'N U T, 0, 0, 0',
	X = 1237.345  mm,	Y = 34.354  mm,	Z = -240.917  mm,
	W = 0.000 deg,	P = 30.000 deg,	R = -176.541 deg
};
P[259]{
   GP1:
	UF : 0, UT : 1,		CONFIG : 'N U T, 0, 0, 0',
	X = 1237.224  mm,	Y = 36.350  mm,	Z = -240.884  mm,
	W = 0.000 deg,	P = 30.000 deg,	R = -176.541 deg
};
P[260]{
   GP1:
	UF : 0, UT : 1,		CONFIG : 'N U T, 0, 0, 0',
	X = 1237.104  mm,	Y = 38.347  mm,	Z = -240.851  mm,
	W = 0.000 deg,	P = 30.000 deg,	R = -176.541 deg
};
P[261]{
   GP1:
	UF : 0, UT : 1,		CONFIG : 'N U T, 0, 0, 0',
	X = 1236.983  mm,	Y = 40.343  mm,	Z = -240.819  mm,
	W = 0.000 deg,	P = 30.000 deg,	R = -176.541 deg
};
P[262]{
   GP1:
	UF : 0, UT : 1,		CONFIG : 'N U T, 0, 0, 0',
	X = 1236.862  mm,	Y = 42.339  mm,	Z = -240.786  mm,
	W = 0.000 deg,	P = 30.000 deg,	R = -176.541 deg
};
P[263]{
   GP1:
	UF : 0, UT : 1,		CONFIG : 'N U T, 0, 0, 0',
	X = 1236.742  mm,	Y = 44.335  mm,	Z = -240.753  mm,
	W = 0.000 deg,	P = 30.000 deg,	R = -176.541 deg
};
P[264]{
   GP1:
	UF : 0, UT : 1,		CONFIG : 'N U T, 0, 0, 0',
	X = 1236.621  mm,	Y = 46.331  mm,	Z = -240.720  mm,
	W = 0.000 deg,	P = 30.000 deg,	R = -176.541 deg
};
P[265]{
   GP1:
	UF : 0, UT : 1,		CONFIG : 'N U T, 0, 0, 0',
	X = 1236.501  mm,	Y = 48.327  mm,	Z = -240.687  mm,
	W = 0.000 deg,	P = 30.000 deg,	R = -176.541 deg
};
P[266]{
   GP1:
	UF : 0, UT : 1,		CONFIG : 'N U T, 0, 0, 0',
	X = 1236.380  mm,	Y = 50.323  mm,	Z = -240.654  mm,
	W = 0.000 deg,	P = 30.000 deg,	R = -176.541 deg
};
P[267]{
   GP1:
	UF : 0, UT : 1,		CONFIG : 'N U T, 0, 0, 0',
	X = 1236.259  mm,	Y = 52.319  mm,	Z = -240.622  mm,
	W = 0.000 deg,	P = 30.000 deg,	R = -176.541 deg
};
P[268]{
   GP1:
	UF : 0, UT : 1,		CONFIG : 'N U T, 0, 0, 0',
	X = 1236.139  mm,	Y = 54.315  mm,	Z = -240.589  mm,
	W = 0.000 deg,	P = 30.000 deg,	R = -176.541 deg
};
P[269]{
   GP1:
	UF : 0, UT : 1,		CONFIG : 'N U T, 0, 0, 0',
	X = 1236.018  mm,	Y = 56.311  mm,	Z = -240.556  mm,
	W = 0.000 deg,	P = 30.000 deg,	R = -176.541 deg
};
P[270]{
   GP1:
	UF : 0, UT : 1,		CONFIG : 'N U T, 0, 0, 0',
	X = 1235.897  mm,	Y = 58.307  mm,	Z = -240.523  mm,
	W = 0.000 deg,	P = 30.000 deg,	R = -176.541 deg
};
P[271]{
   GP1:
	UF : 0, UT : 1,		CONFIG : 'N U T, 0, 0, 0',
	X = 1235.777  mm,	Y = 60.304  mm,	Z = -240.490  mm,
	W = 0.000 deg,	P = 30.000 deg,	R = -176.541 deg
};
P[272]{
   GP1:
	UF : 0, UT : 1,		CONFIG : 'N U T, 0, 0, 0',
	X = 1235.656  mm,	Y = 62.300  mm,	Z = -240.457  mm,
	W = 0.000 deg,	P = 30.000 deg,	R = -176.541 deg
};
P[273]{
   GP1:
	UF : 0, UT : 1,		CONFIG : 'N U T, 0, 0, 0',
	X = 1235.535  mm,	Y = 64.296  mm,	Z = -240.424  mm,
	W = 0.000 deg,	P = 30.000 deg,	R = -176.541 deg
};
P[274]{
   GP1:
	UF : 0, UT : 1,		CONFIG : 'N U T, 0, 0, 0',
	X = 1235.415  mm,	Y = 66.292  mm,	Z = -240.392  mm,
	W = 0.000 deg,	P = 30.000 deg,	R = -176.541 deg
};
P[275]{
   GP1:
	UF : 0, UT : 1,		CONFIG : 'N U T, 0, 0, 0',
	X = 1235.294  mm,	Y = 68.288  mm,	Z = -240.359  mm,
	W = 0.000 deg,	P = 30.000 deg,	R = -176.541 deg
};
P[276]{
   GP1:
	UF : 0, UT : 1,		CONFIG : 'N U T, 0, 0, 0',
	X = 1235.174  mm,	Y = 70.284  mm,	Z = -240.326  mm,
	W = 0.000 deg,	P = 30.000 deg,	R = -176.541 deg
};
P[277]{
   GP1:
	UF : 0, UT : 1,		CONFIG : 'N U T, 0, 0, 0',
	X = 1235.053  mm,	Y = 72.280  mm,	Z = -240.293  mm,
	W = 0.000 deg,	P = 30.000 deg,	R = -165.395 deg
};
P[278]{
   GP1:
	UF : 0, UT : 1,		CONFIG : 'N U T, 0, 0, 0',
	X = 1234.932  mm,	Y = 74.276  mm,	Z = -240.260  mm,
	W = 0.000 deg,	P = 30.000 deg,	R = -157.009 deg
};
P[279]{
   GP1:
	UF : 0, UT : 1,		CONFIG : 'N U T, 0, 0, 0',
	X = 1234.812  mm,	Y = 76.272  mm,	Z = -240.227  mm,
	W = 0.000 deg,	P = 30.000 deg,	R = -148.623 deg
};
P[280]{
   GP1:
	UF : 0, UT : 1,		CONFIG : 'N U T, 0, 0, 0',
	X = 1234.691  mm,	Y = 78.268  mm,	Z = -240.195  mm,
	W = 0.000 deg,	P = 30.000 deg,	R = -140.237 deg
};
P[281]{
   GP1:
	UF : 0, UT : 1,		CONFIG : 'N U T, 0, 0, 0',
	X = 1234.570  mm,	Y = 80.264  mm,	Z = -240.162  mm,
	W = 0.000 deg,	P = 30.000 deg,	R = -134.611 deg
};
P[282]{
   GP1:
	UF : 0, UT : 1,		CONFIG : 'N U T, 0, 0, 0',
	X = 1235.280  mm,	Y = 78.028  mm,	Z = -240.144  mm,
	W = 0.000 deg,	P = 30.000 deg,	R = -134.611 deg
};
P[283]{
   GP1:
	UF : 0, UT : 1,		CONFIG : 'N U T, 0, 0, 0',
	X = 1236.805  mm,	Y = 75.459  mm,	Z = -240.000  mm,
	W = 0.000 deg,	P = 30.000 deg,	R = -134.611 deg
};
P[284]{
   GP1:
	UF : 0, UT : 1,		CONFIG : 'N U T, 0, 0, 0',
	X = 1235.398  mm,	Y = 76.847  mm,	Z = -239.691  mm,
	W = 0.000 deg,	P = 30.000 deg,	R = -134.611 deg
};
P[285]{
   GP1:
	UF : 0, UT : 1,		CONFIG : 'N U T, 0, 0, 0',
	X = 1233.991  mm,	Y = 78.235  mm,	Z = -239.383  mm,
	W = 0.000 deg,	P = 30.000 deg,	R = -134.611 deg
};
P[286]{
   GP1:
	UF : 0, UT : 1,		CONFIG : 'N U T, 0, 0, 0',
	X = 1232.585  mm,	Y = 79.623  mm,	Z = -239.074  mm,
	W = 0.000 deg,	P = 30.000 deg,	R = -134.611 deg
};
P[287]{
   GP1:
	UF : 0, UT : 1,		CONFIG : 'N U T, 0, 0, 0',
	X = 1231.178  mm,	Y = 81.010  mm,	Z = -238.766  mm,
	W = 0.000 deg,	P = 30.000 deg,	R = -134.611 deg
};
P[288]{
   GP1:
	UF : 0, UT : 1,		CONFIG : 'N U T, 0, 0, 0',
	X = 1229.771  mm,	Y = 82.398  mm,	Z = -238.457  mm,
	W = 0.000 deg,	P = 30.000 deg,	R = -134.611 deg
};
P[289]{
   GP1:
	UF : 0, UT : 1,		CONFIG : 'N U T, 0, 0, 0',
	X = 1228.364  mm,	Y = 83.786  mm,	Z = -238.148  mm,
	W = 0.000 deg,	P = 30.000 deg,	R = -134.611 deg
};
P[290]{
   GP1:
	UF : 0, UT : 1,		CONFIG : 'N U T, 0, 0, 0',
	X = 1226.958  mm,	Y = 85.174  mm,	Z = -237.840  mm,
	W = 0.000 deg,	P = 30.000 deg,	R = -134.611 deg
};
P[291]{
   GP1:
	UF : 0, UT : 1,		CONFIG : 'N U T, 0, 0, 0',
	X = 1225.551  mm,	Y = 86.561  mm,	Z = -237.531  mm,
	W = 0.000 deg,	P = 30.000 deg,	R = -134.611 deg
};
P[292]{
   GP1:
	UF : 0, UT : 1,		CONFIG : 'N U T, 0, 0, 0',
	X = 1224.144  mm,	Y = 87.949  mm,	Z = -237.223  mm,
	W = 0.000 deg,	P = 30.000 deg,	R = -134.611 deg
};
P[293]{
   GP1:
	UF : 0, UT : 1,		CONFIG : 'N U T, 0, 0, 0',
	X = 1222.737  mm,	Y = 89.337  mm,	Z = -236.914  mm,
	W = 0.000 deg,	P = 30.000 deg,	R = -134.611 deg
};
P[294]{
   GP1:
	UF : 0, UT : 1,		CONFIG : 'N U T, 0, 0, 0',
	X = 1221.331  mm,	Y = 90.725  mm,	Z = -236.606  mm,
	W = 0.000 deg,	P = 30.000 deg,	R = -134.611 deg
};
P[295]{
   GP1:
	UF : 0, UT : 1,		CONFIG : 'N U T, 0, 0, 0',
	X = 1219.924  mm,	Y = 92.113  mm,	Z = -236.297  mm,
	W = 0.000 deg,	P = 30.000 deg,	R = -134.611 deg
};
P[296]{
   GP1:
	UF : 0, UT : 1,		CONFIG : 'N U T, 0, 0, 0',
	X = 1218.517  mm,	Y = 93.500  mm,	Z = -235.989  mm,
	W = 0.000 deg,	P = 30.000 deg,	R = -134.611 deg
};
P[297]{
   GP1:
	UF : 0, UT : 1,		CONFIG : 'N U T, 0, 0, 0',
	X = 1217.111  mm,	Y = 94.888  mm,	Z = -235.680  mm,
	W = 0.000 deg,	P = 30.000 deg,	R = -134.611 deg
};
P[298]{
   GP1:
	UF : 0, UT : 1,		CONFIG : 'N U T, 0, 0, 0',
	X = 1215.704  mm,	Y = 96.276  mm,	Z = -235.372  mm,
	W = 0.000 deg,	P = 30.000 deg,	R = -134.611 deg
};
P[299]{
   GP1:
	UF : 0, UT : 1,		CONFIG : 'N U T, 0, 0, 0',
	X = 1214.297  mm,	Y = 97.664  mm,	Z = -235.063  mm,
	W = 0.000 deg,	P = 30.000 deg,	R = -134.611 deg
};
P[300]{
   GP1:
	UF : 0, UT : 1,		CONFIG : 'N U T, 0, 0, 0',
	X = 1212.890  mm,	Y = 99.051  mm,	Z = -234.755  mm,
	W = 0.000 deg,	P = 30.000 deg,	R = -134.611 deg
};
P[301]{
   GP1:
	UF : 0, UT : 1,		CONFIG : 'N U T, 0, 0, 0',
	X = 1211.484  mm,	Y = 100.439  mm,	Z = -234.446  mm,
	W = 0.000 deg,	P = 30.000 deg,	R = -134.611 deg
};
P[302]{
   GP1:
	UF : 0, UT : 1,		CONFIG : 'N U T, 0, 0, 0',
	X = 1210.077  mm,	Y = 101.827  mm,	Z = -234.138  mm,
	W = 0.000 deg,	P = 30.000 deg,	R = -134.611 deg
};
P[303]{
   GP1:
	UF : 0, UT : 1,		CONFIG : 'N U T, 0, 0, 0',
	X = 1208.670  mm,	Y = 103.215  mm,	Z = -233.829  mm,
	W = 0.000 deg,	P = 30.000 deg,	R = -134.611 deg
};
P[304]{
   GP1:
	UF : 0, UT : 1,		CONFIG : 'N U T, 0, 0, 0',
	X = 1207.263  mm,	Y = 104.602  mm,	Z = -233.521  mm,
	W = 0.000 deg,	P = 30.000 deg,	R = -147.657 deg
};
P[305]{
   GP1:
	UF : 0, UT : 1,		CONFIG : 'N U T, 0, 0, 0',
	X = 1205.857  mm,	Y = 105.990  mm,	Z = -233.212  mm,
	W = 0.000 deg,	P = 30.000 deg,	R = -156.535 deg
};
P[306]{
   GP1:
	UF : 0, UT : 1,		CONFIG : 'N U T, 0, 0, 0',
	X = 1204.450  mm,	Y = 107.378  mm,	Z = -232.904  mm,
	W = 0.000 deg,	P = 30.000 deg,	R = -165.414 deg
};
P[307]{
   GP1:
	UF : 0, UT : 1,		CONFIG : 'N U T, 0, 0, 0',
	X = 1203.043  mm,	Y = 108.766  mm,	Z = -232.595  mm,
	W = 0.000 deg,	P = 30.000 deg,	R = -174.292 deg
};
P[308]{
   GP1:
	UF : 0, UT : 1,		CONFIG : 'N U T, 0, 0, 0',
	X = 1201.636  mm,	Y = 110.154  mm,	Z = -232.287  mm,
	W = 0.000 deg,	P = 30.000 deg,	R = -179.003 deg
};
P[309]{
   GP1:
	UF : 0, UT : 1,		CONFIG : 'N U T, 0, 0, 0',
	X = 1198.581  mm,	Y = 114.826  mm,	Z = -232.171  mm,
	W = 0.000 deg,	P = 30.000 deg,	R = -179.003 deg
};
P[310]{
   GP1:
	UF : 0, UT : 1,		CONFIG : 'N U T, 0, 0, 0',
	X = 1198.111  mm,	Y = 118.868  mm,	Z = -232.166  mm,
	W = 0.000 deg,	P = 30.000 deg,	R = -179.003 deg
};
P[311]{
   GP1:
	UF : 0, UT : 1,		CONFIG : 'N U T, 0, 0, 0',
	X = 1198.076  mm,	Y = 120.868  mm,	Z = -232.159  mm,
	W = 0.000 deg,	P = 30.000 deg,	R = -179.003 deg
};
P[312]{
   GP1:
	UF : 0, UT : 1,		CONFIG : 'N U T, 0, 0, 0',
	X = 1198.041  mm,	Y = 122.868  mm,	Z = -232.151  mm,
	W = 0.000 deg,	P = 30.000 deg,	R = -179.003 deg
};
P[313]{
   GP1:
	UF : 0, UT : 1,		CONFIG : 'N U T, 0, 0, 0',
	X = 1198.006  mm,	Y = 124.867  mm,	Z = -232.144  mm,
	W = 0.000 deg,	P = 30.000 deg,	R = -179.003 deg
};
P[314]{
   GP1:
	UF : 0, UT : 1,		CONFIG : 'N U T, 0, 0, 0',
	X = 1197.972  mm,	Y = 126.867  mm,	Z = -232.136  mm,
	W = 0.000 deg,	P = 30.000 deg,	R = -179.003 deg
};
P[315]{
   GP1:
	UF : 0, UT : 1,		CONFIG : 'N U T, 0, 0, 0',
	X = 1197.937  mm,	Y = 128.867  mm,	Z = -232.129  mm,
	W = 0.000 deg,	P = 30.000 deg,	R = -179.003 deg
};
P[316]{
   GP1:
	UF : 0, UT : 1,		CONFIG : 'N U T, 0, 0, 0',
	X = 1197.902  mm,	Y = 130.866  mm,	Z = -232.121  mm,
	W = 0.000 deg,	P = 30.000 deg,	R = -179.003 deg
};
P[317]{
   GP1:
	UF : 0, UT : 1,		CONFIG : 'N U T, 0, 0, 0',
	X = 1197.867  mm,	Y = 132.866  mm,	Z = -232.114  mm,
	W = 0.000 deg,	P = 30.000 deg,	R = -179.003 deg
};
P[318]{
   GP1:
	UF : 0, UT : 1,		CONFIG : 'N U T, 0, 0, 0',
	X = 1197.832  mm,	Y = 134.866  mm,	Z = -232.106  mm,
	W = 0.000 deg,	P = 30.000 deg,	R = -179.003 deg
};
P[319]{
   GP1:
	UF : 0, UT : 1,		CONFIG : 'N U T, 0, 0, 0',
	X = 1197.798  mm,	Y = 136.865  mm,	Z = -232.099  mm,
	W = 0.000 deg,	P = 30.000 deg,	R = -179.003 deg
};
P[320]{
   GP1:
	UF : 0, UT : 1,		CONFIG : 'N U T, 0, 0, 0',
	X = 1197.763  mm,	Y = 138.865  mm,	Z = -232.091  mm,
	W = 0.000 deg,	P = 30.000 deg,	R = -179.003 deg
};
P[321]{
   GP1:
	UF : 0, UT : 1,		CONFIG : 'N U T, 0, 0, 0',
	X = 1197.728  mm,	Y = 140.865  mm,	Z = -232.084  mm,
	W = 0.000 deg,	P = 30.000 deg,	R = -179.003 deg
};
P[322]{
   GP1:
	UF : 0, UT : 1,		CONFIG : 'N U T, 0, 0, 0',
	X = 1197.693  mm,	Y = 142.865  mm,	Z = -232.076  mm,
	W = 0.000 deg,	P = 30.000 deg,	R = -179.003 deg
};
P[323]{
   GP1:
	UF : 0, UT : 1,		CONFIG : 'N U T, 0, 0, 0',
	X = 1197.658  mm,	Y = 144.864  mm,	Z = -232.069  mm,
	W = 0.000 deg,	P = 30.000 deg,	R = -179.003 deg
};
P[324]{
   GP1:
	UF : 0, UT : 1,		CONFIG : 'N U T, 0, 0, 0',
	X = 1197.624  mm,	Y = 146.864  mm,	Z = -232.061  mm,
	W = 0.000 deg,	P = 30.000 deg,	R = -179.003 deg
};
P[325]{
   GP1:
	UF : 0, UT : 1,		CONFIG : 'N U T, 0, 0, 0',
	X = 1197.589  mm,	Y = 148.864  mm,	Z = -232.054  mm,
	W = 0.000 deg,	P = 30.000 deg,	R = -179.003 deg
};
P[326]{
   GP1:
	UF : 0, UT : 1,		CONFIG : 'N U T, 0, 0, 0',
	X = 1197.554  mm,	Y = 150.863  mm,	Z = -232.046  mm,
	W = 0.000 deg,	P = 30.000 deg,	R = -179.003 deg
};
P[327]{
   GP1:
	UF : 0, UT : 1,		CONFIG : 'N U T, 0, 0, 0',
	X = 1197.519  mm,	Y = 152.863  mm,	Z = -232.039  mm,
	W = 0.000 deg,	P = 30.000 deg,	R = -179.003 deg
};
P[328]{
   GP1:
	UF : 0, UT : 1,		CONFIG : 'N U T, 0, 0, 0',
	X = 1197.484  mm,	Y = 154.863  mm,	Z = -232.031  mm,
	W = 0.000 deg,	P = 30.000 deg,	R = -179.003 deg
};
P[329]{
   GP1:
	UF : 0, UT : 1,		CONFIG : 'N U T, 0, 0, 0',
	X = 1197.450  mm,	Y = 156.862  mm,	Z = -232.024  mm,
	W = 0.000 deg,	P = 30.000 deg,	R = -179.003 deg
};
P[330]{
   GP1:
	UF : 0, UT : 1,		CONFIG : 'N U T, 0, 0, 0',
	X = 1197.415  mm,	Y = 158.862  mm,	Z = -232.016  mm,
	W = 0.000 deg,	P = 30.000 deg,	R = -179.003 deg
};
P[331]{
   GP1:
	UF : 0, UT : 1,		CONFIG : 'N U T, 0, 0, 0',
	X = 1197.380  mm,	Y = 160.862  mm,	Z = -232.008  mm,
	W = 0.000 deg,	P = 30.000 deg,	R = -179.003 deg
};
P[332]{
   GP1:
	UF : 0, UT : 1,		CONFIG : 'N U T, 0, 0, 0',
	X = 1197.345  mm,	Y = 162.861  mm,	Z = -232.001  mm,
	W = 0.000 deg,	P = 30.000 deg,	R = -179.003 deg
};
P[333]{
   GP1:
	UF : 0, UT : 1,		CONFIG : 'N U T, 0, 0, 0',
	X = 1197.310  mm,	Y = 164.861  mm,	Z = -231.993  mm,
	W = 0.000 deg,	P = 30.000 deg,	R = -179.003 deg
};
P[334]{
   GP1:
	UF : 0, UT : 1,		CONFIG : 'N U T, 0, 0, 0',
	X = 1197.276  mm,	Y = 166.861  mm,	Z = -231.986  mm,
	W = 0.000 deg,	P = 30.000 deg,	R = 175.489 deg
};
P[335]{
   GP1:
	UF : 0, UT : 1,		CONFIG : 'N U T, 0, 0, 0',
	X = 1197.241  mm,	Y = 168.860  mm,	Z = -231.978  mm,
	W = 0.000 deg,	P = 30.000 deg,	R = 166.669 deg
};
P[336]{
   GP1:
	UF : 0, UT : 1,		CONFIG : 'N U T, 0, 0, 0',
	X = 1197.206  mm,	Y = 170.860  mm,	Z = -231.971  mm,
	W = 0.000 deg,	P = 30.000 deg,	R = 157.849 deg
};
P[337]{
   GP1:
	UF : 0, UT : 1,		CONFIG : 'N U T, 0, 0, 0',
	X = 1197.171  mm,	Y = 172.860  mm,	Z = -231.963  mm,
	W = 0.000 deg,	P = 30.000 deg,	R = 149.029 deg
};
P[338]{
   GP1:
	UF : 0, UT : 1,		CONFIG : 'N U T, 0, 0, 0',
	X = 1197.136  mm,	Y = 174.859  mm,	Z = -231.956  mm,
	W = 0.000 deg,	P = 30.000 deg,	R = 140.210 deg
};
P[339]{
   GP1:
	UF : 0, UT : 1,		CONFIG : 'N U T, 0, 0, 0',
	X = 1197.493  mm,	Y = 178.983  mm,	Z = -231.951  mm,
	W = 0.000 deg,	P = 30.000 deg,	R = 136.898 deg
};
P[340]{
   GP1:
	UF : 0, UT : 1,		CONFIG : 'N U T, 0, 0, 0',
	X = 1200.339  mm,	Y = 183.650  mm,	Z = -232.066  mm,
	W = 0.000 deg,	P = 30.000 deg,	R = 136.898 deg
};
P[341]{
   GP1:
	UF : 0, UT : 1,		CONFIG : 'N U T, 0, 0, 0',
	X = 1201.691  mm,	Y = 185.094  mm,	Z = -232.359  mm,
	W = 0.000 deg,	P = 30.000 deg,	R = 136.898 deg
};
P[342]{
   GP1:
	UF : 0, UT : 1,		CONFIG : 'N U T, 0, 0, 0',
	X = 1203.043  mm,	Y = 186.539  mm,	Z = -232.652  mm,
	W = 0.000 deg,	P = 30.000 deg,	R = 136.898 deg
};
P[343]{
   GP1:
	UF : 0, UT : 1,		CONFIG : 'N U T, 0, 0, 0',
	X = 1204.395  mm,	Y = 187.983  mm,	Z = -232.945  mm,
	W = 0.000 deg,	P = 30.000 deg,	R = 136.898 deg
};
P[344]{
   GP1:
	UF : 0, UT : 1,		CONFIG : 'N U T, 0, 0, 0',
	X = 1205.747  mm,	Y = 189.428  mm,	Z = -233.238  mm,
	W = 0.000 deg,	P = 30.000 deg,	R = 136.898 deg
};
P[345]{
   GP1:
	UF : 0, UT : 1,		CONFIG : 'N U T, 0, 0, 0',
	X = 1207.099  mm,	Y = 190.872  mm,	Z = -233.531  mm,
	W = 0.000 deg,	P = 30.000 deg,	R = 136.898 deg
};
P[346]{
   GP1:
	UF : 0, UT : 1,		CONFIG : 'N U T, 0, 0, 0',
	X = 1208.451  mm,	Y = 192.317  mm,	Z = -233.824  mm,
	W = 0.000 deg,	P = 30.000 deg,	R = 136.898 deg
};
P[347]{
   GP1:
	UF : 0, UT : 1,		CONFIG : 'N U T, 0, 0, 0',
	X = 1209.802  mm,	Y = 193.761  mm,	Z = -234.117  mm,
	W = 0.000 deg,	P = 30.000 deg,	R = 136.898 deg
};
P[348]{
   GP1:
	UF : 0, UT : 1,		CONFIG : 'N U T, 0, 0, 0',
	X = 1211.154  mm,	Y = 195.206  mm,	Z = -234.410  mm,
	W = 0.000 deg,	P = 30.000 deg,	R = 136.898 deg
};
P[349]{
   GP1:
	UF : 0, UT : 1,		CONFIG : 'N U T, 0, 0, 0',
	X = 1212.506  mm,	Y = 196.650  mm,	Z = -234.703  mm,
	W = 0.000 deg,	P = 30.000 deg,	R = 136.898 deg
};
P[350]{
   GP1:
	UF : 0, UT : 1,		CONFIG : 'N U T, 0, 0, 0',
	X = 1213.858  mm,	Y = 198.095  mm,	Z = -234.996  mm,
	W = 0.000 deg,	P = 30.000 deg,	R = 136.898 deg
};
P[351]{
   GP1:
	UF : 0, UT : 1,		CONFIG : 'N U T, 0, 0, 0',
	X = 1215.210  mm,	Y = 199.539  mm,	Z = -235.289  mm,
	W = 0.000 deg,	P = 30.000 deg,	R = 136.898 deg
};
P[352]{
   GP1:
	UF : 0, UT : 1,		CONFIG : 'N U T, 0, 0, 0',
	X = 1216.562  mm,	Y = 200.984  mm,	Z = -235.582  mm,
	W = 0.000 deg,	P = 30.000 deg,	R = 136.898 deg
};
P[353]{
   GP1:
	UF : 0, UT : 1,		CONFIG : 'N U T, 0, 0, 0',
	X = 1217.914  mm,	Y = 202.428  mm,	Z = -235.875  mm,
	W = 0.000 deg,	P = 30.000 deg,	R = 136.898 deg
};
P[354]{
   GP1:
	UF : 0, UT : 1,		CONFIG : 'N U T, 0, 0, 0',
	X = 1219.265  mm,	Y = 203.873  mm,	Z = -236.168  mm,
	W = 0.000 deg,	P = 30.000 deg,	R = 136.898 deg
};
P[355]{
   GP1:
	UF : 0, UT : 1,		CONFIG : 'N U T, 0, 0, 0',
	X = 1220.617  mm,	Y = 205.317  mm,	Z = -236.461  mm,
	W = 0.000 deg,	P = 30.000 deg,	R = 136.898 deg
};
P[356]{
   GP1:
	UF : 0, UT : 1,		CONFIG : 'N U T, 0, 0, 0',
	X = 1221.969  mm,	Y = 206.762  mm,	Z = -236.754  mm,
	W = 0.000 deg,	P = 30.000 deg,	R = 136.898 deg
};
P[357]{
   GP1:
	UF : 0, UT : 1,		CONFIG : 'N U T, 0, 0, 0',
	X = 1223.321  mm,	Y = 208.207  mm,	Z = -237.047  mm,
	W = 0.000 deg,	P = 30.000 deg,	R = 136.898 deg
};
P[358]{
   GP1:
	UF : 0, UT : 1,		CONFIG : 'N U T, 0, 0, 0',
	X = 1224.673  mm,	Y = 209.651  mm,	Z = -237.340  mm,
	W = 0.000 deg,	P = 30.000 deg,	R = 136.898 deg
};
P[359]{
   GP1:
	UF : 0, UT : 1,		CONFIG : 'N U T, 0, 0, 0',
	X = 1226.025  mm,	Y = 211.096  mm,	Z = -237.633  mm,
	W = 0.000 deg,	P = 30.000 deg,	R = 136.898 deg
};
P[360]{
   GP1:
	UF : 0, UT : 1,		CONFIG : 'N U T, 0, 0, 0',
	X = 1227.377  mm,	Y = 212.540  mm,	Z = -237.926  mm,
	W = 0.000 deg,	P = 30.000 deg,	R = 149.041 deg
};
P[361]{
   GP1:
	UF : 0, UT : 1,		CONFIG : 'N U T, 0, 0, 0',
	X = 1228.728  mm,	Y = 213.985  mm,	Z = -238.219  mm,
	W = 0.000 deg,	P = 30.000 deg,	R = 157.776 deg
};
P[362]{
   GP1:
	UF : 0, UT : 1,		CONFIG : 'N U T, 0, 0, 0',
	X = 1230.080  mm,	Y = 215.429  mm,	Z = -238.512  mm,
	W = 0.000 deg,	P = 30.000 deg,	R = 166.512 deg
};
P[363]{
   GP1:
	UF : 0, UT : 1,		CONFIG : 'N U T, 0, 0, 0',
	X = 1231.432  mm,	Y = 216.874  mm,	Z = -238.805  mm,
	W = 0.000 deg,	P = 30.000 deg,	R = 175.248 deg
};
P[364]{
   GP1:
	UF : 0, UT : 1,		CONFIG : 'N U T, 0, 0, 0',
	X = 1232.784  mm,	Y = 218.318  mm,	Z = -239.098  mm,
	W = 0.000 deg,	P = 30.000 deg,	R = -179.424 deg
};
P[365]{
   GP1:
	UF : 0, UT : 1,		CONFIG : 'N U T, 0, 0, 0',
	X = 1231.909  mm,	Y = 216.731  mm,	Z = -239.275  mm,
	W = 0.000 deg,	P = 30.000 deg,	R = -179.424 deg
};
P[366]{
   GP1:
	UF : 0, UT : 1,		CONFIG : 'N U T, 0, 0, 0',
	X = 1230.895  mm,	Y = 213.049  mm,	Z = -239.274  mm,
	W = 0.000 deg,	P = 30.000 deg,	R = -179.424 deg
};
P[367]{
   GP1:
	UF : 0, UT : 1,		CONFIG : 'N U T, 0, 0, 0',
	X = 1230.875  mm,	Y = 215.049  mm,	Z = -239.272  mm,
	W = 0.000 deg,	P = 30.000 deg,	R = -179.424 deg
};
P[368]{
   GP1:
	UF : 0, UT : 1,		CONFIG : 'N U T, 0, 0, 0',
	X = 1230.855  mm,	Y = 217.049  mm,	Z = -239.269  mm,
	W = 0.000 deg,	P = 30.000 deg,	R = -179.424 deg
};
P[369]{
   GP1:
	UF : 0, UT : 1,		CONFIG : 'N U T, 0, 0, 0',
	X = 1230.835  mm,	Y = 219.048  mm,	Z = -239.267  mm,
	W = 0.000 deg,	P = 30.000 deg,	R = -179.424 deg
};
P[370]{
   GP1:
	UF : 0, UT : 1,		CONFIG : 'N U T, 0, 0, 0',
	X = 1230.814  mm,	Y = 221.048  mm,	Z = -239.265  mm,
	W = 0.000 deg,	P = 30.000 deg,	R = -179.424 deg
};
P[371]{
   GP1:
	UF : 0, UT : 1,		CONFIG : 'N U T, 0, 0, 0',
	X = 1230.802  mm,	Y = 222.257  mm,	Z = -239.263  mm,
	W = 0.000 deg,	P = 30.000 deg,	R = -179.424 deg
};
/END
